C05468=1078.580,132.841,429.704,174.173,23.522,154.056
C05469=1078.585,133.090,429.683,174.174,23.524,154.056
C05470=1078.591,133.339,429.663,174.176,23.527,154.057
C05471=1078.596,133.588,429.643,174.178,23.529,154.057
C05472=1078.602,133.837,429.624,174.180,23.532,154.057
C05473=1078.607,134.086,429.603,174.181,23.533,154.057
C05474=1078.613,134.335,429.583,174.184,23.536,154.058
C05475=1078.619,134.584,429.563,174.186,23.538,154.058
C05476=1078.625,134.833,429.543,174.187,23.541,154.058
C05477=1078.630,135.083,429.522,174.190,23.543,154.058
C05478=1078.636,135.332,429.502,174.191,23.545,154.058
C05479=1078.642,135.581,429.482,174.193,23.548,154.058
C05480=1078.647,135.830,429.462,174.195,23.550,154.059
C05481=1078.653,136.079,429.442,174.197,23.552,154.059
C05482=1078.659,136.328,429.421,174.198,23.555,154.059
C05483=1078.664,136.578,429.402,174.201,23.557,154.059
C05484=1078.670,136.827,429.382,174.203,23.559,154.059
C05485=1078.676,137.075,429.362,174.204,23.561,154.060
C05486=1078.681,137.325,429.341,174.207,23.564,154.060
C05487=1078.687,137.574,429.321,174.208,23.566,154.060
C05488=1078.693,137.823,429.300,174.210,23.568,154.060
C05489=1078.699,138.072,429.280,174.212,23.571,154.061
C05490=1078.704,138.321,429.260,174.214,23.573,154.061
C05491=1078.710,138.570,429.240,174.215,23.575,154.061
C05492=1078.715,138.819,429.219,174.218,23.577,154.061
C05493=1078.720,139.068,429.199,174.220,23.580,154.061
C05494=1078.727,139.318,429.178,174.221,23.582,154.062
C05495=1078.732,139.567,429.158,174.224,23.584,154.062
C05496=1078.738,139.816,429.138,174.225,23.587,154.062
C05497=1078.744,140.065,429.117,174.228,23.589,154.062
C05498=1078.750,140.314,429.097,174.229,23.591,154.063
C05499=1078.755,140.563,429.077,174.231,23.594,154.063
C05500=1078.760,140.812,429.056,174.233,23.596,154.063
C05501=1078.767,141.061,429.036,174.235,23.598,154.063
C05502=1078.772,141.310,429.015,174.237,23.601,154.063
C05503=1078.777,141.560,428.995,174.239,23.603,154.064
C05504=1078.783,141.808,428.975,174.241,23.605,154.064
C05505=1078.788,142.058,428.954,174.243,23.608,154.064
C05506=1078.794,142.307,428.934,174.244,23.610,154.064
C05507=1078.800,142.557,428.913,174.247,23.612,154.064
C05508=1078.806,142.805,428.893,174.248,23.615,154.065
C05509=1078.812,143.086,428.869,174.251,23.617,154.065
C05510=1078.818,143.367,428.846,174.253,23.620,154.065
C05511=1078.824,143.647,428.824,174.255,23.622,154.065
C05512=1078.831,143.928,428.800,174.257,23.625,154.066
C05513=1078.836,144.177,428.779,174.260,23.627,154.066
C05514=1078.842,144.427,428.758,174.261,23.629,154.066
C05515=1078.848,144.675,428.738,174.263,23.632,154.066
C05516=1078.853,144.925,428.718,174.265,23.634,154.066
C05517=1078.859,145.173,428.697,174.267,23.637,154.067
C05518=1078.864,145.422,428.676,174.269,23.639,154.067
C05519=1078.871,145.672,428.656,174.271,23.641,154.067
C05520=1078.876,145.921,428.635,174.273,23.643,154.067
C05521=1078.881,146.169,428.614,174.274,23.645,154.067
C05522=1078.887,146.418,428.593,174.277,23.648,154.068
C05523=1078.893,146.668,428.573,174.279,23.650,154.068
C05524=1078.898,146.917,428.552,174.281,23.652,154.068
C05525=1078.904,147.166,428.531,174.283,23.655,154.068
C05526=1078.910,147.415,428.510,174.285,23.657,154.068
C05527=1078.916,147.664,428.490,174.286,23.659,154.069
C05528=1078.921,147.913,428.470,174.289,23.662,154.069
C05529=1078.927,148.162,428.448,174.290,23.663,154.069
C05530=1078.933,148.412,428.428,174.293,23.666,154.069
C05531=1078.938,148.661,428.407,174.295,23.668,154.069
C05532=1078.943,148.909,428.386,174.296,23.671,154.070
C05533=1078.949,149.158,428.365,174.299,23.673,154.070
C05534=1078.955,149.408,428.345,174.301,23.675,154.070
C05535=1078.961,149.656,428.324,174.302,23.677,154.070
C05536=1078.966,149.906,428.303,174.305,23.680,154.070
C05537=1078.972,150.155,428.281,174.306,23.682,154.071
C05538=1078.977,150.404,428.261,174.308,23.684,154.071
C05539=1078.983,150.653,428.240,174.311,23.687,154.071
C05540=1078.989,150.902,428.219,174.312,23.689,154.071
C05541=1078.994,151.151,428.198,174.314,23.691,154.071
C05542=1079.000,151.400,428.177,174.317,23.694,154.072
C05543=1079.005,151.649,428.156,174.318,23.696,154.072
C05544=1079.011,151.898,428.135,174.321,23.698,154.072
C05545=1079.016,152.147,428.114,174.323,23.701,154.072
C05546=1079.022,152.396,428.093,174.324,23.702,154.072
C05547=1079.028,152.646,428.072,174.326,23.705,154.073
C05548=1079.033,152.894,428.051,174.328,23.707,154.073
C05549=1079.039,153.143,428.030,174.330,23.709,154.073
C05550=1079.045,153.392,428.008,174.333,23.712,154.073
C05551=1079.050,153.642,427.988,174.334,23.714,154.073
C05552=1079.056,153.890,427.967,174.336,23.716,154.073
C05553=1079.061,154.140,427.946,174.339,23.719,154.074
C05554=1079.067,154.388,427.924,174.340,23.721,154.074
C05555=1079.073,154.638,427.904,174.342,23.723,154.074
C05556=1079.078,154.887,427.882,174.345,23.726,154.074
C05557=1079.084,155.135,427.861,174.346,23.727,154.074
C05558=1079.090,155.385,427.840,174.349,23.730,154.075
C05559=1079.095,155.634,427.819,174.351,23.732,154.075
C05560=1079.101,155.883,427.798,174.352,23.734,154.075
C05561=1079.107,156.132,427.777,174.354,23.737,154.075
C05562=1079.112,156.380,427.755,174.357,23.739,154.075
C05563=1079.117,156.631,427.734,174.358,23.741,154.076
C05564=1079.123,156.879,427.713,174.361,23.744,154.076
C05565=1079.129,157.128,427.691,174.363,23.746,154.076
C05566=1079.134,157.377,427.670,174.364,23.748,154.076
C05567=1079.140,157.626,427.649,174.367,23.751,154.076
C05568=1079.146,157.875,427.627,174.369,23.753,154.077
C05569=1079.151,158.124,427.607,174.371,23.755,154.077
C05570=1079.157,158.374,427.585,174.373,23.757,154.077
C05571=1079.162,158.622,427.563,174.375,23.760,154.077
C05572=1079.168,158.871,427.542,174.377,23.762,154.077
C05573=1079.175,159.152,427.518,174.380,23.764,154.078
C05574=1079.181,159.432,427.494,174.382,23.767,154.078
C05575=1079.187,159.712,427.471,174.384,23.769,154.078
C05576=1079.193,159.993,427.446,174.387,23.772,154.078
C05577=1079.199,160.242,427.425,174.388,23.774,154.078
C05578=1079.205,160.491,427.403,174.390,23.777,154.079
C05579=1079.211,160.740,427.382,174.393,23.779,154.079
C05580=1079.216,160.989,427.361,174.395,23.781,154.079
C05581=1079.222,161.238,427.339,174.396,23.784,154.079
C05582=1079.227,161.487,427.318,174.399,23.786,154.079
C05583=1079.233,161.736,427.296,174.401,23.788,154.080
C05584=1079.238,161.985,427.274,174.402,23.790,154.080
C05585=1079.244,162.234,427.253,174.405,23.793,154.080
C05586=1079.249,162.483,427.231,174.407,23.795,154.080
C05587=1079.255,162.732,427.209,174.409,23.797,154.080
C05588=1079.260,162.982,427.188,174.411,23.800,154.081
C05589=1079.265,163.230,427.167,174.413,23.802,154.081
C05590=1079.271,163.480,427.145,174.415,23.805,154.081
C05591=1079.276,163.728,427.123,174.417,23.807,154.081
C05592=1079.282,163.977,427.102,174.419,23.809,154.081
C05593=1079.287,164.226,427.080,174.422,23.812,154.082
C05594=1079.293,164.475,427.058,174.424,23.814,154.082
C05595=1079.298,164.724,427.036,174.425,23.816,154.082
C05596=1079.304,164.973,427.015,174.428,23.818,154.082
C05597=1079.309,165.222,426.993,174.430,23.821,154.082
C05598=1079.315,165.471,426.971,174.432,23.823,154.083
C05599=1079.320,165.721,426.949,174.434,23.825,154.083
C05600=1079.326,165.969,426.928,174.436,23.828,154.083
C05601=1079.331,166.219,426.906,174.438,23.830,154.083
C05602=1079.337,166.467,426.884,174.440,23.832,154.083
C05603=1079.342,166.717,426.862,174.442,23.835,154.084
C05604=1079.347,166.965,426.840,174.444,23.837,154.084
C05605=1079.353,167.215,426.819,174.447,23.840,154.084
C05606=1079.358,167.463,426.797,174.448,23.841,154.084
C05607=1079.364,167.712,426.774,174.450,23.844,154.084
C05608=1079.369,167.961,426.752,174.453,23.846,154.085
C05609=1079.375,168.210,426.731,174.455,23.848,154.085
C05610=1079.380,168.459,426.709,174.457,23.851,154.085
C05611=1079.386,168.708,426.687,174.459,23.853,154.085
C05612=1079.391,168.957,426.665,174.461,23.855,154.085
C05613=1079.397,169.206,426.644,174.464,23.858,154.086
C05614=1079.403,169.456,426.622,174.466,23.860,154.086
C05615=1079.408,169.704,426.599,174.467,23.863,154.086
C05616=1079.414,169.953,426.577,174.470,23.865,154.086
C05617=1079.419,170.202,426.556,174.472,23.867,154.086
C05618=1079.425,170.451,426.534,174.474,23.870,154.087
C05619=1079.431,170.700,426.512,174.476,23.871,154.087
C05620=1079.436,170.948,426.490,174.478,23.874,154.087
C05621=1079.442,171.198,426.467,174.480,23.876,154.087
C05622=1079.447,171.447,426.446,174.483,23.879,154.087
C05623=1079.453,171.696,426.424,174.484,23.880,154.087
C05624=1079.459,171.945,426.401,174.487,23.883,154.088
C05625=1079.464,172.193,426.380,174.489,23.885,154.088
C05626=1079.470,172.443,426.358,174.491,23.888,154.088
C05627=1079.475,172.691,426.335,174.494,23.890,154.088
C05628=1079.481,172.940,426.313,174.495,23.892,154.088
C05629=1079.486,173.190,426.291,174.497,23.894,154.089
C05630=1079.491,173.438,426.268,174.500,23.897,154.089
C05631=1079.498,173.687,426.247,174.502,23.899,154.089
C05632=1079.503,173.937,426.225,174.504,23.901,154.089
C05633=1079.509,174.185,426.203,174.506,23.903,154.089
C05634=1079.514,174.434,426.180,174.508,23.905,154.089
C05635=1079.520,174.684,426.158,174.511,23.908,154.090
C05636=1079.526,174.932,426.136,174.513,23.910,154.090
C05637=1079.532,175.212,426.111,174.515,23.913,154.090
C05638=1079.538,175.492,426.086,174.518,23.915,154.090
C05639=1079.545,175.773,426.061,174.520,23.918,154.091
C05640=1079.551,176.053,426.036,174.522,23.920,154.091
C05641=1079.557,176.302,426.013,174.525,23.922,154.091
C05642=1079.562,176.550,425.992,174.527,23.925,154.091
C05643=1079.568,176.800,425.969,174.529,23.927,154.091
C05644=1079.573,177.049,425.946,174.532,23.930,154.091
C05645=1079.579,177.298,425.925,174.533,23.931,154.092
C05646=1079.585,177.546,425.902,174.535,23.934,154.092
C05647=1079.590,177.795,425.880,174.538,23.936,154.092
C05648=1079.597,178.044,425.858,174.540,23.939,154.092
C05649=1079.602,178.293,425.835,174.543,23.941,154.092
C05650=1079.607,178.542,425.813,174.545,23.943,154.092
C05651=1079.614,178.790,425.791,174.546,23.945,154.093
C05652=1079.619,179.040,425.768,174.549,23.947,154.093
C05653=1079.625,179.289,425.745,174.551,23.950,154.093
C05654=1079.630,179.538,425.723,174.554,23.952,154.093
C05655=1079.636,179.786,425.701,174.556,23.955,154.093
C05656=1079.642,180.035,425.678,174.558,23.957,154.093
C05657=1079.647,180.285,425.656,174.560,23.959,154.094
C05658=1079.654,180.533,425.634,174.562,23.961,154.094
C05659=1079.659,180.783,425.611,174.564,23.963,154.094
C05660=1079.665,181.032,425.588,174.567,23.966,154.094
C05661=1079.670,181.280,425.566,174.569,23.968,154.094
C05662=1079.676,181.529,425.544,174.571,23.970,154.094
C05663=1079.682,181.778,425.521,174.574,23.972,154.095
C05664=1079.688,182.027,425.498,174.575,23.974,154.095
C05665=1079.693,182.276,425.476,174.578,23.976,154.095
C05666=1079.699,182.525,425.454,174.580,23.979,154.095
C05667=1079.705,182.774,425.431,174.582,23.981,154.095
C05668=1079.710,183.022,425.408,174.585,23.983,154.095
C05669=1079.716,183.271,425.386,174.587,23.986,154.096
C05670=1079.721,183.520,425.363,174.590,23.988,154.096
C05671=1079.728,183.769,425.341,174.592,23.990,154.096
C05672=1079.734,184.018,425.318,174.594,23.992,154.096
C05673=1079.739,184.267,425.296,174.596,23.995,154.096
C05674=1079.745,184.516,425.273,174.598,23.997,154.096
C05675=1079.751,184.765,425.250,174.601,23.999,154.097
C05676=1079.757,185.014,425.227,174.603,24.001,154.097
C05677=1079.763,185.263,425.204,174.605,24.003,154.097
C05678=1079.767,185.511,425.181,174.608,24.006,154.097
C05679=1079.773,185.761,425.159,174.610,24.008,154.097
C05680=1079.778,186.010,425.136,174.611,24.011,154.098
C05681=1079.784,186.258,425.113,174.614,24.013,154.098
C05682=1079.790,186.507,425.090,174.616,24.015,154.098
C05683=1079.795,186.756,425.068,174.618,24.018,154.098
C05684=1079.800,187.005,425.044,174.621,24.020,154.098
C05685=1079.806,187.254,425.021,174.623,24.023,154.099
C05686=1079.811,187.503,424.998,174.625,24.025,154.099
C05687=1079.817,187.751,424.975,174.628,24.027,154.099
C05688=1079.823,188.000,424.952,174.630,24.030,154.099
C05689=1079.827,188.249,424.929,174.633,24.032,154.099
C05690=1079.833,188.498,424.906,174.634,24.034,154.099
C05691=1079.839,188.747,424.883,174.636,24.036,154.100
C05692=1079.844,188.996,424.860,174.639,24.039,154.100
C05693=1079.850,189.244,424.837,174.641,24.041,154.100
C05694=1079.855,189.494,424.814,174.643,24.044,154.100
C05695=1079.861,189.743,424.791,174.646,24.046,154.100
C05696=1079.867,189.991,424.768,174.648,24.048,154.101
C05697=1079.872,190.240,424.745,174.650,24.051,154.101
C05698=1079.877,190.488,424.722,174.653,24.053,154.101
C05699=1079.882,190.738,424.699,174.655,24.055,154.101
C05700=1079.888,190.987,424.676,174.657,24.058,154.101
C05701=1079.895,191.267,424.650,174.660,24.060,154.102
C05702=1079.901,191.546,424.624,174.662,24.063,154.102
C05703=1079.907,191.827,424.597,174.665,24.066,154.102
C05704=1079.913,192.106,424.571,174.668,24.068,154.102
C05705=1079.919,192.355,424.548,174.670,24.070,154.102
C05706=1079.925,192.604,424.526,174.672,24.073,154.103
C05707=1079.930,192.853,424.502,174.675,24.075,154.103
C05708=1079.936,193.101,424.478,174.677,24.077,154.103
C05709=1079.941,193.350,424.455,174.679,24.080,154.103
C05710=1079.947,193.599,424.432,174.681,24.082,154.103
C05711=1079.952,193.848,424.409,174.683,24.084,154.103
C05712=1079.958,194.097,424.386,174.686,24.087,154.104
C05713=1079.964,194.345,424.362,174.688,24.089,154.104
C05714=1079.969,194.595,424.339,174.690,24.091,154.104
C05715=1079.975,194.844,424.316,174.693,24.093,154.104
C05716=1079.980,195.092,424.293,174.695,24.096,154.104
C05717=1079.986,195.341,424.269,174.697,24.098,154.105
C05718=1079.991,195.590,424.246,174.700,24.100,154.105
C05719=1079.997,195.839,424.223,174.702,24.103,154.105
C05720=1080.003,196.087,424.199,174.704,24.105,154.105
C05721=1080.008,196.336,424.175,174.707,24.107,154.105
C05722=1080.014,196.585,424.153,174.709,24.110,154.105
C05723=1080.020,196.833,424.129,174.712,24.112,154.106
C05724=1080.025,197.083,424.105,174.714,24.114,154.106
C05725=1080.031,197.332,424.082,174.716,24.117,154.106
C05726=1080.037,197.581,424.058,174.719,24.119,154.106
C05727=1080.042,197.830,424.035,174.721,24.121,154.106
C05728=1080.048,198.079,424.012,174.723,24.124,154.107
C05729=1080.054,198.327,423.988,174.726,24.126,154.107
C05730=1080.059,198.576,423.965,174.728,24.128,154.107
C05731=1080.065,198.824,423.941,174.731,24.131,154.107
C05732=1080.071,199.073,423.918,174.733,24.133,154.107
C05733=1080.076,199.322,423.894,174.735,24.135,154.107
C05734=1080.082,199.571,423.871,174.738,24.137,154.108
C05735=1080.087,199.821,423.847,174.740,24.140,154.108
C05736=1080.093,200.069,423.823,174.742,24.142,154.108
C05737=1080.099,200.318,423.800,174.745,24.144,154.108
C05738=1080.104,200.566,423.776,174.747,24.147,154.108
C05739=1080.110,200.815,423.753,174.749,24.149,154.108
C05740=1080.116,201.064,423.729,174.752,24.151,154.109
C05741=1080.122,201.313,423.705,174.754,24.154,154.109
C05742=1080.128,201.562,423.682,174.757,24.156,154.109
C05743=1080.133,201.810,423.658,174.759,24.159,154.109
C05744=1080.139,202.059,423.635,174.761,24.161,154.109
C05745=1080.144,202.308,423.610,174.764,24.163,154.109
C05746=1080.151,202.557,423.587,174.766,24.165,154.110
C05747=1080.156,202.806,423.563,174.768,24.168,154.110
C05748=1080.162,203.054,423.539,174.771,24.170,154.110
C05749=1080.167,203.304,423.516,174.773,24.172,154.110
C05750=1080.173,203.552,423.492,174.776,24.175,154.110
C05751=1080.178,203.800,423.468,174.778,24.177,154.111
C05752=1080.184,204.050,423.444,174.780,24.179,154.111
C05753=1080.190,204.299,423.420,174.783,24.182,154.111
C05754=1080.195,204.547,423.396,174.785,24.184,154.111
C05755=1080.200,204.796,423.372,174.787,24.186,154.111
C05756=1080.206,205.045,423.349,174.791,24.189,154.112
C05757=1080.211,205.293,423.324,174.793,24.192,154.112
C05758=1080.217,205.543,423.300,174.795,24.194,154.112
C05759=1080.223,205.791,423.277,174.798,24.196,154.112
C05760=1080.228,206.040,423.253,174.800,24.199,154.112
C05761=1080.234,206.289,423.228,174.803,24.201,154.112
C05762=1080.240,206.538,423.204,174.805,24.203,154.113
C05763=1080.245,206.787,423.181,174.807,24.206,154.113
C05764=1080.251,207.035,423.157,174.809,24.208,154.113
C05765=1080.274,208.069,423.057,174.909,24.261,154.111
C05766=1080.283,208.468,423.017,174.913,24.267,154.112
C05767=1080.292,208.867,422.978,174.917,24.272,154.113
C05768=1080.302,209.266,422.939,174.921,24.277,154.113
C05769=1080.311,209.665,422.899,174.924,24.282,154.114
C05770=1080.317,209.914,422.874,174.926,24.286,154.114
C05771=1080.322,210.163,422.850,174.929,24.289,154.115
C05772=1080.328,210.411,422.825,174.931,24.293,154.115
C05773=1080.334,210.660,422.800,174.934,24.296,154.116
C05774=1080.339,210.909,422.776,174.936,24.299,154.116
C05775=1080.345,211.157,422.751,174.938,24.303,154.116
C05776=1080.351,211.406,422.726,174.940,24.306,154.117
C05777=1080.356,211.655,422.702,174.943,24.309,154.117
C05778=1080.362,211.904,422.677,174.945,24.313,154.118
C05779=1080.368,212.152,422.652,174.947,24.316,154.118
C05780=1080.373,212.401,422.626,174.949,24.319,154.118
C05781=1080.378,212.650,422.602,174.952,24.323,154.119
C05782=1080.385,212.899,422.577,174.954,24.326,154.119
C05783=1080.391,213.148,422.552,174.957,24.329,154.120
C05784=1080.396,213.396,422.528,174.959,24.332,154.120
C05785=1080.402,213.645,422.503,174.961,24.336,154.121
C05786=1080.407,213.894,422.478,174.964,24.340,154.121
C05787=1080.413,214.143,422.452,174.966,24.343,154.121
C05788=1080.418,214.391,422.427,174.968,24.346,154.122
C05789=1080.424,214.640,422.403,174.970,24.349,154.122
C05790=1080.430,214.888,422.378,174.973,24.353,154.122
C05791=1080.436,215.137,422.353,174.975,24.356,154.123
C05792=1080.441,215.385,422.328,174.977,24.359,154.123
C05793=1080.447,215.635,422.303,174.979,24.362,154.124
C05794=1080.453,215.883,422.278,174.982,24.366,154.124
C05795=1080.458,216.131,422.253,174.984,24.370,154.125
C05796=1080.464,216.381,422.228,174.986,24.373,154.125
C05797=1080.469,216.629,422.203,174.989,24.376,154.125
C05798=1080.475,216.878,422.178,174.992,24.380,154.126
C05799=1080.481,217.127,422.153,174.994,24.383,154.126
C05800=1080.486,217.375,422.127,174.996,24.386,154.127
C05801=1080.492,217.624,422.102,174.998,24.389,154.127
C05802=1080.498,217.872,422.077,175.001,24.393,154.127
C05803=1080.504,218.121,422.052,175.003,24.396,154.128
C05804=1080.509,218.370,422.026,175.005,24.399,154.128
C05805=1080.515,218.619,422.002,175.007,24.402,154.129
C05806=1080.521,218.867,421.977,175.010,24.406,154.129
C05807=1080.526,219.116,421.951,175.013,24.409,154.129
C05808=1080.532,219.364,421.926,175.015,24.412,154.130
C05809=1080.538,219.614,421.901,175.018,24.416,154.130
C05810=1080.544,219.862,421.876,175.020,24.420,154.131
C05811=1080.549,220.111,421.850,175.022,24.423,154.131
C05812=1080.555,220.359,421.825,175.024,24.426,154.132
C05813=1080.561,220.608,421.799,175.027,24.430,154.132
C05814=1080.567,220.857,421.774,175.029,24.433,154.132
C05815=1080.572,221.105,421.749,175.031,24.436,154.133
C05816=1080.578,221.354,421.724,175.033,24.439,154.133
C05817=1080.584,221.603,421.698,175.036,24.443,154.133
C05818=1080.593,222.006,421.657,175.040,24.448,154.134
C05819=1080.602,222.409,421.615,175.044,24.453,154.135
C05820=1080.612,222.813,421.574,175.048,24.459,154.135
C05821=1080.621,223.215,421.533,175.052,24.464,154.136
C05822=1080.626,223.464,421.507,175.054,24.467,154.136
C05823=1080.632,223.713,421.482,175.057,24.471,154.137
C05824=1080.637,223.961,421.456,175.059,24.474,154.137
C05825=1080.643,224.210,421.431,175.061,24.478,154.138
C05826=1080.649,224.459,421.405,175.064,24.481,154.138
C05827=1080.655,224.707,421.379,175.066,24.484,154.139
C05828=1080.660,224.956,421.354,175.068,24.488,154.139
C05829=1080.666,225.204,421.328,175.071,24.491,154.139
C05830=1080.672,225.453,421.303,175.073,24.494,154.140
C05831=1080.677,225.702,421.277,175.075,24.498,154.140
C05832=1080.683,225.950,421.252,175.078,24.501,154.141
C05833=1080.688,226.199,421.226,175.081,24.504,154.141
C05834=1080.694,226.448,421.200,175.083,24.508,154.142
C05835=1080.700,226.697,421.174,175.085,24.511,154.142
C05836=1080.706,226.945,421.148,175.088,24.515,154.142
C05837=1080.711,227.193,421.123,175.090,24.518,154.143
C05838=1080.717,227.442,421.097,175.092,24.521,154.143
C05839=1080.723,227.691,421.072,175.095,24.525,154.143
C05840=1080.728,227.940,421.046,175.097,24.528,154.144
C05841=1080.735,228.188,421.020,175.099,24.531,154.144
C05842=1080.740,228.437,420.994,175.102,24.535,154.145
C05843=1080.746,228.686,420.968,175.105,24.538,154.145
C05844=1080.751,228.934,420.943,175.107,24.541,154.145
C05845=1080.757,229.182,420.916,175.110,24.545,154.146
C05846=1080.763,229.431,420.890,175.112,24.548,154.146
C05847=1080.769,229.680,420.865,175.114,24.551,154.147
C05848=1080.774,229.929,420.839,175.117,24.554,154.147
C05849=1080.780,230.177,420.812,175.119,24.558,154.147
C05850=1080.786,230.426,420.787,175.121,24.561,154.148
C05851=1080.792,230.675,420.761,175.124,24.564,154.148
C05852=1080.797,230.922,420.735,175.127,24.568,154.149
C05853=1080.802,231.171,420.709,175.129,24.571,154.149
C05854=1080.809,231.420,420.683,175.132,24.575,154.150
C05855=1080.814,231.668,420.657,175.134,24.578,154.150
C05856=1080.820,231.917,420.631,175.136,24.581,154.150
C05857=1080.826,232.166,420.604,175.139,24.585,154.151
C05858=1080.831,232.415,420.578,175.141,24.588,154.151
C05859=1080.837,232.663,420.552,175.143,24.591,154.152
C05860=1080.843,232.912,420.526,175.146,24.595,154.152
C05861=1080.849,233.160,420.500,175.148,24.598,154.152
C05862=1080.854,233.409,420.474,175.151,24.601,154.153
C05863=1080.859,233.657,420.448,175.154,24.605,154.153
C05864=1080.865,233.906,420.421,175.156,24.608,154.154
C05865=1080.871,234.154,420.395,175.159,24.612,154.154
C05866=1080.876,234.403,420.369,175.161,24.615,154.154
C05867=1080.882,234.651,420.342,175.163,24.618,154.155
C05868=1080.888,234.900,420.317,175.166,24.622,154.155
C05869=1080.894,235.148,420.290,175.168,24.625,154.156
C05870=1080.903,235.543,420.248,175.172,24.630,154.156
C05871=1080.911,235.938,420.207,175.176,24.636,154.157
C05872=1080.921,236.333,420.165,175.180,24.641,154.158
C05873=1080.930,236.728,420.122,175.184,24.646,154.158
C05874=1080.935,236.976,420.096,175.187,24.650,154.159
C05875=1080.941,237.225,420.070,175.189,24.653,154.159
C05876=1080.947,237.474,420.043,175.192,24.657,154.160
C05877=1080.952,237.722,420.017,175.194,24.660,154.160
C05878=1080.958,237.971,419.991,175.196,24.663,154.160
C05879=1080.964,238.219,419.964,175.199,24.667,154.161
C05880=1080.969,238.468,419.937,175.201,24.670,154.161
C05881=1080.975,238.716,419.911,175.204,24.673,154.162
C05882=1080.981,238.965,419.885,175.206,24.677,154.162
C05883=1080.986,239.213,419.858,175.209,24.680,154.162
C05884=1080.992,239.462,419.831,175.212,24.683,154.163
C05885=1080.998,239.710,419.805,175.214,24.686,154.163
C05886=1081.004,239.958,419.778,175.217,24.690,154.164
C05887=1081.009,240.207,419.752,175.219,24.694,154.164
C05888=1081.016,240.456,419.725,175.221,24.697,154.165
C05889=1081.021,240.705,419.699,175.224,24.700,154.165
C05890=1081.027,240.953,419.672,175.226,24.704,154.165
C05891=1081.033,241.201,419.645,175.229,24.707,154.166
C05892=1081.038,241.450,419.618,175.231,24.710,154.166
C05893=1081.044,241.698,419.591,175.234,24.714,154.166
C05894=1081.050,241.947,419.565,175.237,24.717,154.167
C05895=1081.055,242.195,419.538,175.239,24.720,154.167
C05896=1081.061,242.444,419.511,175.242,24.724,154.168
C05897=1081.067,242.693,419.484,175.244,24.727,154.168
C05898=1081.073,242.941,419.458,175.247,24.730,154.168
C05899=1081.078,243.190,419.431,175.249,24.734,154.169
C05900=1081.084,243.438,419.404,175.252,24.738,154.169
C05901=1081.090,243.686,419.377,175.254,24.741,154.170
C05902=1081.096,243.935,419.351,175.256,24.744,154.170
C05903=1081.101,244.183,419.323,175.260,24.747,154.171
C05904=1081.106,244.432,419.297,175.262,24.751,154.171
C05905=1081.113,244.681,419.270,175.265,24.755,154.172
C05906=1081.118,244.930,419.242,175.267,24.758,154.172
C05907=1081.124,245.178,419.216,175.270,24.761,154.172
C05908=1081.129,245.426,419.189,175.272,24.764,154.173
C05909=1081.134,245.675,419.162,175.274,24.768,154.173
C05910=1081.140,245.923,419.135,175.277,24.771,154.174
C05911=1081.147,246.172,419.108,175.279,24.775,154.174
C05912=1081.152,246.420,419.080,175.282,24.778,154.174
C05913=1081.158,246.669,419.054,175.284,24.781,154.175
C05914=1081.163,246.917,419.027,175.288,24.785,154.175
C05915=1081.168,247.166,419.000,175.290,24.788,154.176
C05916=1081.175,247.413,418.972,175.293,24.792,154.176
C05917=1081.180,247.663,418.945,175.295,24.795,154.177
C05918=1081.186,247.911,418.918,175.297,24.799,154.177
C05919=1081.191,248.160,418.891,175.300,24.802,154.177
C05920=1081.197,248.408,418.864,175.302,24.805,154.178
C05921=1081.202,248.656,418.836,175.305,24.809,154.178
C05922=1081.211,249.044,418.794,175.309,24.814,154.179
C05923=1081.220,249.432,418.752,175.313,24.820,154.180
C05924=1081.228,249.820,418.709,175.317,24.825,154.180
C05925=1081.238,250.208,418.666,175.321,24.830,154.181
C05926=1081.243,250.457,418.639,175.324,24.834,154.181
C05927=1081.249,250.705,418.611,175.326,24.837,154.182
C05928=1081.254,250.954,418.584,175.329,24.841,154.182
C05929=1081.260,251.201,418.557,175.331,24.844,154.183
C05930=1081.266,251.451,418.529,175.334,24.848,154.183
C05931=1081.271,251.700,418.502,175.336,24.851,154.184
C05932=1081.277,251.947,418.474,175.339,24.855,154.184
C05933=1081.282,252.196,418.447,175.341,24.858,154.184
C05934=1081.289,252.444,418.419,175.344,24.862,154.185
C05935=1081.294,252.693,418.392,175.347,24.865,154.185
C05936=1081.299,252.941,418.364,175.350,24.869,154.186
C05937=1081.306,253.190,418.337,175.352,24.872,154.186
C05938=1081.311,253.438,418.309,175.355,24.875,154.186
C05939=1081.317,253.686,418.282,175.357,24.878,154.187
C05940=1081.323,253.935,418.254,175.360,24.883,154.187
C05941=1081.328,254.183,418.226,175.362,24.886,154.188
C05942=1081.334,254.432,418.200,175.365,24.889,154.188
C05943=1081.340,254.681,418.171,175.367,24.892,154.189
C05944=1081.345,254.929,418.143,175.370,24.896,154.189
C05945=1081.351,255.177,418.117,175.373,24.899,154.189
C05946=1081.357,255.426,418.088,175.376,24.903,154.190
C05947=1081.363,255.673,418.061,175.378,24.906,154.190
C05948=1081.368,255.922,418.034,175.381,24.910,154.191
C05949=1081.374,256.171,418.005,175.383,24.913,154.191
C05950=1081.380,256.419,417.978,175.386,24.916,154.191
C05951=1081.386,256.668,417.950,175.388,24.920,154.192
C05952=1081.391,256.916,417.922,175.391,24.923,154.192
C05953=1081.397,257.164,417.895,175.393,24.927,154.193
C05954=1081.403,257.412,417.867,175.396,24.930,154.193
C05955=1081.408,257.661,417.840,175.399,24.933,154.194
C05956=1081.414,257.910,417.811,175.402,24.937,154.194
C05957=1081.420,258.158,417.784,175.404,24.940,154.195
C05958=1081.426,258.406,417.756,175.407,24.944,154.195
C05959=1081.431,258.654,417.728,175.409,24.947,154.195
C05960=1081.438,258.903,417.700,175.412,24.951,154.196
C05961=1081.443,259.152,417.673,175.415,24.954,154.196
C05962=1081.449,259.400,417.644,175.417,24.957,154.197
C05963=1081.454,259.648,417.616,175.420,24.961,154.197
C05964=1081.461,259.897,417.589,175.423,24.964,154.197
C05965=1081.466,260.145,417.561,175.426,24.968,154.198
C05966=1081.472,260.394,417.532,175.428,24.971,154.198
C05967=1081.478,260.642,417.504,175.431,24.975,154.199
C05968=1081.484,260.890,417.477,175.433,24.978,154.199
C05969=1081.490,261.138,417.449,175.436,24.982,154.200
C05970=1081.496,261.387,417.420,175.438,24.985,154.200
C05971=1081.501,261.635,417.392,175.441,24.988,154.200
C05972=1081.508,261.883,417.365,175.444,24.992,154.201
C05973=1081.513,262.131,417.337,175.447,24.995,154.201
C05974=1081.522,262.517,417.293,175.451,25.001,154.202
C05975=1081.531,262.903,417.249,175.455,25.006,154.202
C05976=1081.540,263.287,417.205,175.459,25.011,154.203
C05977=1081.550,263.673,417.162,175.463,25.016,154.204
C05978=1081.556,263.921,417.134,175.466,25.020,154.204
C05979=1081.561,264.169,417.106,175.468,25.023,154.205
C05980=1081.567,264.418,417.078,175.471,25.026,154.205
C05981=1081.573,264.666,417.049,175.474,25.030,154.206
C05982=1081.579,264.914,417.021,175.477,25.034,154.206
C05983=1081.584,265.162,416.993,175.480,25.037,154.206
C05984=1081.590,265.411,416.964,175.482,25.041,154.207
C05985=1081.596,265.659,416.936,175.485,25.044,154.207
C05986=1081.602,265.907,416.907,175.487,25.047,154.208
C05987=1081.607,266.156,416.879,175.490,25.051,154.208
C05988=1081.612,266.404,416.851,175.492,25.054,154.209
C05989=1081.618,266.653,416.822,175.495,25.058,154.209
C05990=1081.624,266.901,416.794,175.498,25.062,154.209
C05991=1081.630,267.149,416.765,175.500,25.065,154.210
C05992=1081.636,267.398,416.736,175.504,25.069,154.210
C05993=1081.641,267.646,416.708,175.506,25.072,154.211
C05994=1081.647,267.894,416.680,175.509,25.076,154.211
C05995=1081.653,268.142,416.651,175.512,25.079,154.212
C05996=1081.659,268.390,416.623,175.514,25.083,154.212
C05997=1081.665,268.639,416.595,175.517,25.086,154.213
C05998=1081.670,268.887,416.565,175.519,25.089,154.213
C05999=1081.676,269.136,416.537,175.522,25.093,154.213
C06000=1081.682,269.384,416.508,175.525,25.097,154.214
C06001=1081.687,269.632,416.480,175.527,25.100,154.214
C06002=1081.693,269.880,416.451,175.531,25.103,154.215
C06003=1081.699,270.129,416.423,175.533,25.107,154.215
C06004=1081.704,270.377,416.393,175.536,25.111,154.216
C06005=1081.710,270.625,416.365,175.539,25.115,154.216
C06006=1081.716,270.873,416.336,175.541,25.118,154.217
C06007=1081.722,271.121,416.308,175.544,25.121,154.217
C06008=1081.727,271.370,416.278,175.546,25.125,154.217
C06009=1081.733,271.619,416.250,175.549,25.128,154.218
C06010=1081.739,271.867,416.221,175.552,25.132,154.218
C06011=1081.745,272.115,416.193,175.554,25.135,154.219
C06012=1081.750,272.363,416.163,175.558,25.139,154.219
C06013=1081.757,272.611,416.134,175.561,25.142,154.220
C06014=1081.762,272.859,416.106,175.563,25.146,154.220
C06015=1081.767,273.108,416.077,175.566,25.149,154.220
C06016=1081.774,273.356,416.048,175.568,25.153,154.221
C06017=1081.780,273.605,416.019,175.571,25.157,154.221
C06018=1081.785,273.853,415.990,175.574,25.160,154.222
C06019=1081.791,274.101,415.961,175.576,25.164,154.222
C06020=1081.797,274.349,415.932,175.579,25.167,154.223
C06021=1081.802,274.598,415.903,175.582,25.171,154.223
C06022=1081.808,274.845,415.875,175.584,25.174,154.224
C06023=1081.813,275.094,415.845,175.587,25.178,154.224
C06024=1081.820,275.342,415.816,175.591,25.182,154.225
C06025=1081.826,275.591,415.788,175.593,25.185,154.225
C06026=1081.834,275.978,415.742,175.597,25.191,154.226
C06027=1081.843,276.366,415.696,175.602,25.196,154.226
C06028=1081.853,276.755,415.650,175.605,25.202,154.227
C06029=1081.860,277.143,415.605,175.610,25.207,154.228
C06030=1081.867,277.391,415.576,175.613,25.211,154.228
C06031=1081.872,277.640,415.546,175.615,25.214,154.229
C06032=1081.879,277.888,415.517,175.618,25.218,154.229
C06033=1081.883,278.136,415.488,175.621,25.222,154.230
C06034=1081.890,278.384,415.459,175.623,25.226,154.230
C06035=1081.895,278.632,415.429,175.627,25.229,154.231
C06036=1081.901,278.881,415.400,175.630,25.233,154.231
C06037=1081.907,279.129,415.371,175.632,25.236,154.232
C06038=1081.913,279.377,415.342,175.635,25.240,154.232
C06039=1081.919,279.626,415.312,175.638,25.244,154.233
C06040=1081.924,279.873,415.283,175.640,25.247,154.233
C06041=1081.930,280.121,415.254,175.643,25.251,154.233
C06042=1081.935,280.370,415.224,175.646,25.255,154.234
C06043=1081.942,280.618,415.195,175.648,25.258,154.234
C06044=1081.947,280.866,415.165,175.651,25.261,154.235
C06045=1081.954,281.114,415.136,175.654,25.265,154.235
C06046=1081.959,281.362,415.106,175.656,25.269,154.236
C06047=1081.965,281.611,415.076,175.660,25.272,154.236
C06048=1081.971,281.859,415.047,175.663,25.276,154.237
C06049=1081.976,282.107,415.018,175.665,25.279,154.237
C06050=1081.982,282.354,414.988,175.668,25.283,154.238
C06051=1081.987,282.603,414.958,175.671,25.287,154.238
C06052=1081.993,282.851,414.929,175.674,25.291,154.239
C06053=1081.999,283.100,414.899,175.676,25.294,154.239
C06054=1082.004,283.348,414.870,175.679,25.298,154.240
C06055=1082.010,283.596,414.839,175.682,25.302,154.240
C06056=1082.017,283.844,414.810,175.684,25.305,154.241
C06057=1082.022,284.092,414.781,175.687,25.309,154.241
C06058=1082.028,284.340,414.750,175.690,25.313,154.242
C06059=1082.033,284.589,414.721,175.693,25.316,154.242
C06060=1082.039,284.837,414.691,175.696,25.320,154.242
C06061=1082.045,285.085,414.661,175.699,25.324,154.243
C06062=1082.051,285.333,414.632,175.702,25.327,154.243
C06063=1082.056,285.581,414.602,175.704,25.331,154.244
C06064=1082.062,285.829,414.572,175.707,25.335,154.244
C06065=1082.068,286.078,414.542,175.710,25.338,154.245
C06066=1082.074,286.325,414.512,175.713,25.342,154.245
C06067=1082.080,286.574,414.483,175.715,25.345,154.246
C06068=1082.086,286.821,414.452,175.718,25.349,154.246
C06069=1082.091,287.070,414.423,175.721,25.353,154.247
C06070=1082.097,287.318,414.392,175.723,25.356,154.247
C06071=1082.103,287.566,414.363,175.726,25.360,154.248
C06072=1082.109,287.814,414.333,175.729,25.364,154.248
C06073=1082.115,288.062,414.303,175.732,25.368,154.249
C06074=1082.120,288.310,414.273,175.735,25.371,154.249
C06075=1082.126,288.558,414.243,175.738,25.375,154.250
C06076=1082.132,288.806,414.213,175.741,25.379,154.250
C06077=1082.137,289.055,414.183,175.744,25.383,154.251
C06078=1082.147,289.453,414.135,175.748,25.388,154.251
C06079=1082.156,289.850,414.086,175.753,25.395,154.252
C06080=1082.166,290.248,414.038,175.757,25.400,154.253
C06081=1082.174,290.646,413.990,175.762,25.406,154.254
C06082=1082.180,290.894,413.960,175.764,25.410,154.254
C06083=1082.186,291.142,413.929,175.767,25.413,154.255
C06084=1082.192,291.390,413.900,175.770,25.417,154.255
C06085=1082.198,291.639,413.869,175.773,25.421,154.256
C06086=1082.204,291.887,413.839,175.776,25.425,154.256
C06087=1082.210,292.135,413.808,175.778,25.428,154.257
C06088=1082.215,292.382,413.778,175.781,25.432,154.257
C06089=1082.221,292.631,413.748,175.784,25.436,154.258
C06090=1082.227,292.879,413.718,175.787,25.440,154.258
C06091=1082.233,293.126,413.688,175.790,25.443,154.259
C06092=1082.238,293.374,413.657,175.793,25.447,154.259
C06093=1082.244,293.623,413.626,175.796,25.451,154.260
C06094=1082.250,293.871,413.596,175.799,25.455,154.260
C06095=1082.256,294.119,413.565,175.802,25.459,154.261
C06096=1082.261,294.367,413.536,175.804,25.463,154.261
C06097=1082.267,294.615,413.505,175.807,25.466,154.262
C06098=1082.273,294.863,413.475,175.810,25.470,154.262
C06099=1082.279,295.111,413.444,175.813,25.474,154.263
C06100=1082.285,295.359,413.414,175.816,25.478,154.263
C06101=1082.290,295.607,413.383,175.818,25.482,154.264
C06102=1082.296,295.855,413.353,175.821,25.485,154.264
C06103=1082.302,296.103,413.322,175.824,25.489,154.265
C06104=1082.308,296.351,413.292,175.827,25.493,154.265
C06105=1082.313,296.600,413.261,175.830,25.497,154.266
C06106=1082.319,296.847,413.230,175.832,25.500,154.266
C06107=1082.325,297.095,413.199,175.835,25.504,154.267
C06108=1082.332,297.343,413.168,175.838,25.508,154.267
C06109=1082.337,297.591,413.138,175.841,25.512,154.268
C06110=1082.343,297.839,413.107,175.844,25.516,154.268
C06111=1082.348,298.087,413.077,175.847,25.520,154.269
C06112=1082.354,298.336,413.045,175.850,25.524,154.270
C06113=1082.360,298.584,413.015,175.853,25.528,154.270
C06114=1082.365,298.831,412.983,175.856,25.532,154.271
C06115=1082.371,299.079,412.953,175.859,25.536,154.271
C06116=1082.376,299.327,412.922,175.862,25.539,154.272
C06117=1082.383,299.576,412.891,175.864,25.543,154.272
C06118=1082.388,299.823,412.860,175.867,25.547,154.273
C06119=1082.394,300.071,412.829,175.870,25.551,154.273
C06120=1082.399,300.319,412.799,175.873,25.555,154.274
C06121=1082.405,300.567,412.768,175.876,25.559,154.274
C06122=1082.411,300.815,412.736,175.879,25.563,154.275
C06123=1082.417,301.063,412.706,175.881,25.567,154.276
C06124=1082.422,301.311,412.675,175.884,25.571,154.276
C06125=1082.428,301.559,412.643,175.887,25.575,154.277
C06126=1082.433,301.807,412.612,175.890,25.579,154.277
C06127=1082.440,302.054,412.581,175.893,25.582,154.278
C06128=1082.445,302.302,412.550,175.896,25.586,154.278
C06129=1082.451,302.551,412.520,175.899,25.590,154.279
C06130=1082.461,302.963,412.467,175.904,25.597,154.280
C06131=1082.470,303.375,412.416,175.908,25.603,154.280
C06132=1082.479,303.787,412.364,175.913,25.610,154.281
C06133=1082.489,304.199,412.312,175.918,25.616,154.282
C06134=1082.494,304.447,412.281,175.921,25.621,154.283
C06135=1082.501,304.695,412.250,175.924,25.625,154.283
C06136=1082.506,304.943,412.218,175.927,25.629,154.284
C06137=1082.512,305.191,412.188,175.930,25.632,154.285
C06138=1082.518,305.439,412.156,175.933,25.636,154.285
C06139=1082.523,305.687,412.125,175.936,25.640,154.286
C06140=1082.530,305.935,412.093,175.939,25.644,154.286
C06141=1082.535,306.182,412.062,175.941,25.648,154.287
C06142=1082.541,306.431,412.031,175.944,25.652,154.287
C06143=1082.547,306.678,411.999,175.947,25.656,154.288
C06144=1082.552,306.926,411.968,175.950,25.660,154.288
C06145=1082.559,307.174,411.937,175.953,25.664,154.289
C06146=1082.564,307.422,411.905,175.956,25.668,154.290
C06147=1082.570,307.670,411.873,175.959,25.672,154.290
C06148=1082.576,307.917,411.842,175.962,25.676,154.291
C06149=1082.582,308.166,411.811,175.965,25.680,154.291
C06150=1082.587,308.414,411.779,175.968,25.684,154.292
C06151=1082.594,308.662,411.748,175.970,25.688,154.292
C06152=1082.599,308.909,411.716,175.973,25.692,154.293
C06153=1082.605,309.157,411.684,175.976,25.696,154.293
C06154=1082.611,309.405,411.654,175.979,25.700,154.294
C06155=1082.617,309.653,411.622,175.982,25.704,154.294
C06156=1082.623,309.902,411.590,175.985,25.708,154.295
C06157=1082.629,310.149,411.558,175.988,25.712,154.296
C06158=1082.635,310.397,411.526,175.991,25.716,154.296
C06159=1082.641,310.644,411.495,175.994,25.720,154.297
C06160=1082.647,310.893,411.463,175.997,25.724,154.297
C06161=1082.653,311.140,411.432,176.000,25.728,154.298
C06162=1082.659,311.388,411.400,176.003,25.732,154.298
C06163=1082.665,311.636,411.368,176.007,25.736,154.299
C06164=1082.670,311.884,411.336,176.009,25.740,154.300
C06165=1082.677,312.132,411.305,176.012,25.744,154.300
C06166=1082.683,312.380,411.273,176.015,25.748,154.301
C06167=1082.688,312.627,411.241,176.018,25.752,154.301
C06168=1082.694,312.876,411.209,176.021,25.756,154.302
C06169=1082.700,313.124,411.177,176.024,25.760,154.302
C06170=1082.706,313.371,411.146,176.027,25.764,154.303
C06171=1082.712,313.619,411.114,176.030,25.768,154.304
C06172=1082.718,313.867,411.082,176.033,25.772,154.304
C06173=1082.724,314.115,411.050,176.036,25.776,154.305
C06174=1082.730,314.363,411.018,176.039,25.781,154.305
C06175=1082.737,314.610,410.986,176.042,25.785,154.306
C06176=1082.743,314.859,410.954,176.045,25.788,154.306
C06177=1082.748,315.106,410.922,176.048,25.793,154.307
C06178=1082.753,315.355,410.890,176.051,25.797,154.308
C06179=1082.759,315.602,410.858,176.054,25.801,154.308
C06180=1082.765,315.850,410.825,176.057,25.805,154.309
C06181=1082.771,316.098,410.793,176.060,25.810,154.309
C06182=1082.781,316.513,410.739,176.064,25.816,154.310
C06183=1082.790,316.928,410.685,176.069,25.824,154.312
C06184=1082.799,317.344,410.631,176.075,25.831,154.313
C06185=1082.809,317.759,410.577,176.079,25.838,154.314
C06186=1082.814,318.006,410.545,176.082,25.842,154.314
C06187=1082.820,318.254,410.513,176.085,25.846,154.315
C06188=1082.826,318.502,410.481,176.088,25.851,154.315
C06189=1082.832,318.750,410.447,176.091,25.855,154.316
C06190=1082.837,318.998,410.416,176.094,25.859,154.317
C06191=1082.844,319.245,410.383,176.097,25.863,154.317
C06192=1082.849,319.494,410.350,176.100,25.868,154.318
C06193=1082.855,319.741,410.318,176.103,25.872,154.319
C06194=1082.861,319.989,410.286,176.106,25.876,154.319
C06195=1082.867,320.236,410.253,176.109,25.880,154.320
C06196=1082.872,320.485,410.221,176.112,25.885,154.321
C06197=1082.878,320.733,410.188,176.115,25.889,154.321
C06198=1082.884,320.980,410.156,176.118,25.894,154.322
C06199=1082.889,321.228,410.123,176.121,25.897,154.322
C06200=1082.896,321.476,410.090,176.124,25.902,154.323
C06201=1082.902,321.724,410.058,176.127,25.906,154.324
C06202=1082.907,321.972,410.025,176.129,25.911,154.324
C06203=1082.913,322.219,409.993,176.132,25.915,154.325
C06204=1082.919,322.467,409.960,176.136,25.919,154.326
C06205=1082.924,322.715,409.927,176.138,25.923,154.326
C06206=1082.931,322.962,409.894,176.142,25.928,154.327
C06207=1082.937,323.211,409.862,176.145,25.932,154.327
C06208=1082.942,323.458,409.829,176.148,25.937,154.328
C06209=1082.949,323.706,409.796,176.151,25.941,154.329
C06210=1082.955,323.954,409.764,176.154,25.945,154.329
C06211=1082.959,324.201,409.731,176.157,25.949,154.330
C06212=1082.966,324.449,409.698,176.160,25.954,154.331
C06213=1082.972,324.697,409.666,176.163,25.958,154.331
C06214=1082.978,324.945,409.632,176.166,25.962,154.332
C06215=1082.984,325.193,409.600,176.169,25.967,154.333
C06216=1082.989,325.441,409.567,176.172,25.971,154.333
C06217=1082.995,325.688,409.534,176.175,25.976,154.334
C06218=1083.002,325.936,409.501,176.178,25.980,154.335
C06219=1083.007,326.184,409.468,176.181,25.984,154.335
C06220=1083.014,326.431,409.435,176.184,25.989,154.336
C06221=1083.019,326.679,409.402,176.187,25.993,154.337
C06222=1083.025,326.927,409.369,176.190,25.997,154.337
C06223=1083.031,327.175,409.336,176.194,26.002,154.338
C06224=1083.037,327.422,409.303,176.197,26.006,154.339
C06225=1083.044,327.670,409.270,176.200,26.011,154.339
C06226=1083.049,327.918,409.237,176.203,26.015,154.340
C06227=1083.055,328.165,409.204,176.206,26.020,154.341
C06228=1083.061,328.413,409.171,176.209,26.024,154.341
C06229=1083.067,328.661,409.138,176.212,26.028,154.342
C06230=1083.073,328.909,409.105,176.215,26.033,154.343
C06231=1083.079,329.156,409.072,176.217,26.037,154.343
C06232=1083.085,329.405,409.038,176.220,26.041,154.344
C06233=1083.092,329.653,409.006,176.223,26.046,154.344
C06234=1083.101,330.060,408.951,176.229,26.053,154.346
C06235=1083.111,330.469,408.896,176.234,26.061,154.347
C06236=1083.121,330.878,408.841,176.239,26.068,154.348
C06237=1083.131,331.286,408.786,176.244,26.075,154.349
C06238=1083.137,331.534,408.753,176.247,26.080,154.350
C06239=1083.143,331.781,408.720,176.250,26.084,154.350
C06240=1083.149,332.029,408.686,176.253,26.089,154.351
C06241=1083.154,332.277,408.653,176.256,26.093,154.352
C06242=1083.160,332.524,408.619,176.259,26.098,154.352
C06243=1083.167,332.772,408.586,176.262,26.102,154.353
C06244=1083.172,333.020,408.553,176.266,26.107,154.354
C06245=1083.179,333.268,408.518,176.269,26.111,154.354
C06246=1083.184,333.516,408.485,176.272,26.116,154.355
C06247=1083.190,333.764,408.452,176.275,26.121,154.356
C06248=1083.196,334.011,408.418,176.278,26.125,154.357
C06249=1083.202,334.259,408.385,176.281,26.130,154.357
C06250=1083.208,334.506,408.351,176.284,26.135,154.358
C06251=1083.213,334.754,408.317,176.287,26.139,154.359
C06252=1083.220,335.002,408.283,176.290,26.144,154.360
C06253=1083.225,335.250,408.250,176.293,26.149,154.360
C06254=1083.231,335.497,408.216,176.296,26.153,154.361
C06255=1083.238,335.744,408.183,176.299,26.158,154.362
C06256=1083.243,335.992,408.149,176.303,26.163,154.362
C06257=1083.250,336.240,408.115,176.306,26.167,154.363
C06258=1083.255,336.488,408.081,176.309,26.172,154.364
C06259=1083.261,336.735,408.047,176.312,26.176,154.365
C06260=1083.267,336.983,408.014,176.315,26.181,154.365
C06261=1083.273,337.230,407.980,176.318,26.186,154.366
C06262=1083.279,337.478,407.945,176.321,26.191,154.367
C06263=1083.285,337.726,407.912,176.324,26.195,154.367
C06264=1083.291,337.973,407.878,176.327,26.200,154.368
C06265=1083.298,338.221,407.844,176.330,26.205,154.369
C06266=1083.303,338.469,407.811,176.333,26.209,154.370
C06267=1083.308,338.716,407.776,176.337,26.214,154.370
C06268=1083.314,338.964,407.742,176.340,26.219,154.371
C06269=1083.321,339.212,407.708,176.343,26.224,154.372
C06270=1083.326,339.460,407.674,176.346,26.228,154.373
C06271=1083.332,339.707,407.640,176.350,26.233,154.373
C06272=1083.338,339.954,407.606,176.352,26.238,154.374
C06273=1083.344,340.202,407.572,176.355,26.243,154.375
C06274=1083.350,340.449,407.538,176.358,26.248,154.376
C06275=1083.356,340.697,407.504,176.361,26.252,154.376
C06276=1083.363,340.945,407.469,176.365,26.257,154.377
C06277=1083.368,341.192,407.435,176.368,26.262,154.378
C06278=1083.373,341.440,407.401,176.371,26.267,154.379
C06279=1083.380,341.688,407.367,176.374,26.272,154.380
C06280=1083.386,341.936,407.333,176.378,26.277,154.380
C06281=1083.392,342.183,407.299,176.380,26.282,154.381
C06282=1083.398,342.431,407.264,176.383,26.287,154.382
C06283=1083.404,342.678,407.230,176.386,26.292,154.383
C06284=1083.409,342.926,407.196,176.390,26.297,154.384
C06285=1083.416,343.173,407.160,176.393,26.301,154.384
C06286=1083.426,343.576,407.105,176.398,26.309,154.386
C06287=1083.435,343.979,407.049,176.403,26.317,154.387
C06288=1083.444,344.382,406.993,176.408,26.325,154.388
C06289=1083.455,344.784,406.937,176.414,26.333,154.389
C06290=1083.461,345.032,406.902,176.417,26.338,154.390
C06291=1083.466,345.280,406.868,176.419,26.343,154.391
C06292=1083.473,345.528,406.833,176.423,26.349,154.392
C06293=1083.479,345.774,406.799,176.426,26.353,154.393
C06294=1083.484,346.022,406.764,176.429,26.358,154.393
C06295=1083.490,346.270,406.729,176.433,26.363,154.394
C06296=1083.496,346.517,406.695,176.436,26.368,154.395
C06297=1083.502,346.765,406.660,176.438,26.373,154.396
C06298=1083.508,347.012,406.626,176.441,26.378,154.397
C06299=1083.514,347.260,406.591,176.445,26.383,154.397
C06300=1083.520,347.507,406.556,176.448,26.389,154.398
C06301=1083.526,347.755,406.521,176.451,26.393,154.399
C06302=1083.532,348.002,406.486,176.455,26.399,154.400
C06303=1083.538,348.250,406.452,176.458,26.404,154.401
C06304=1083.544,348.497,406.416,176.460,26.409,154.402
C06305=1083.550,348.745,406.382,176.464,26.414,154.402
C06306=1083.555,348.993,406.347,176.467,26.419,154.403
C06307=1083.562,349.240,406.312,176.470,26.424,154.404
C06308=1083.567,349.488,406.277,176.474,26.430,154.405
C06309=1083.574,349.735,406.242,176.477,26.434,154.406
C06310=1083.579,349.982,406.207,176.479,26.440,154.407
C06311=1083.586,350.230,406.173,176.483,26.445,154.408
C06312=1083.591,350.477,406.137,176.486,26.450,154.408
C06313=1083.598,350.725,406.103,176.489,26.455,154.409
C06314=1083.604,350.973,406.067,176.493,26.460,154.410
C06315=1083.610,351.219,406.032,176.496,26.465,154.411
C06316=1083.616,351.468,405.997,176.499,26.471,154.412
C06317=1083.622,351.714,405.962,176.502,26.476,154.413
C06318=1083.628,351.962,405.927,176.505,26.481,154.414
C06319=1083.634,352.210,405.892,176.509,26.487,154.414
C06320=1083.640,352.457,405.857,176.512,26.491,154.415
C06321=1083.646,352.704,405.821,176.515,26.497,154.416
C06322=1083.653,352.952,405.786,176.518,26.502,154.417
C06323=1083.658,353.199,405.751,176.521,26.507,154.418
C06324=1083.664,353.447,405.716,176.525,26.513,154.419
C06325=1083.670,353.694,405.681,176.528,26.518,154.420
C06326=1083.676,353.941,405.645,176.531,26.523,154.421
C06327=1083.682,354.189,405.609,176.534,26.529,154.422
C06328=1083.688,354.436,405.575,176.537,26.534,154.422
C06329=1083.694,354.683,405.539,176.541,26.539,154.423
C06330=1083.700,354.931,405.503,176.544,26.544,154.424
C06331=1083.705,355.179,405.469,176.547,26.550,154.425
C06332=1083.711,355.426,405.433,176.550,26.555,154.426
C06333=1083.718,355.674,405.398,176.553,26.561,154.427
C06334=1083.724,355.921,405.362,176.557,26.566,154.428
C06335=1083.730,356.168,405.327,176.560,26.571,154.429
C06336=1083.736,356.416,405.291,176.563,26.577,154.430
C06337=1083.743,356.663,405.255,176.566,26.582,154.431
C06338=1083.752,357.069,405.197,176.572,26.591,154.432
C06339=1083.762,357.474,405.139,176.576,26.600,154.434
C06340=1083.772,357.880,405.080,176.582,26.609,154.435
C06341=1083.781,358.286,405.022,176.588,26.618,154.437
C06342=1083.788,358.533,404.986,176.590,26.623,154.438
C06343=1083.794,358.781,404.950,176.594,26.629,154.438
C06344=1083.800,359.028,404.914,176.597,26.635,154.440
C06345=1083.806,359.275,404.879,176.601,26.640,154.440
C06346=1083.812,359.522,404.843,176.603,26.645,154.441
C06347=1083.818,359.770,404.807,176.607,26.651,154.442
C06348=1083.824,360.018,404.771,176.610,26.657,154.443
C06349=1083.830,360.265,404.735,176.614,26.662,154.444
C06350=1083.836,360.512,404.699,176.617,26.668,154.445
C06351=1083.842,360.759,404.664,176.620,26.674,154.446
C06352=1083.848,361.006,404.627,176.623,26.679,154.447
C06353=1083.854,361.254,404.591,176.627,26.685,154.448
C06354=1083.861,361.501,404.555,176.630,26.690,154.449
C06355=1083.867,361.749,404.519,176.633,26.696,154.450
C06356=1083.873,361.997,404.484,176.636,26.702,154.451
C06357=1083.878,362.243,404.447,176.640,26.708,154.452
C06358=1083.884,362.491,404.412,176.643,26.713,154.453
C06359=1083.891,362.738,404.375,176.646,26.719,154.454
C06360=1083.897,362.985,404.339,176.649,26.724,154.455
C06361=1083.903,363.232,404.303,176.653,26.730,154.456
C06362=1083.909,363.479,404.267,176.656,26.736,154.457
C06363=1083.915,363.727,404.231,176.659,26.742,154.458
C06364=1083.922,363.974,404.195,176.662,26.747,154.459
C06365=1083.928,364.222,404.159,176.666,26.753,154.460
C06366=1083.933,364.469,404.122,176.669,26.759,154.461
C06367=1083.940,364.716,404.085,176.672,26.765,154.462
C06368=1083.945,364.963,404.049,176.675,26.770,154.463
C06369=1083.952,365.210,404.014,176.679,26.776,154.464
C06370=1083.958,365.457,403.977,176.682,26.782,154.465
C06371=1083.964,365.704,403.941,176.685,26.788,154.466
C06372=1083.970,365.952,403.904,176.689,26.794,154.467
C06373=1083.976,366.199,403.868,176.692,26.799,154.468
C06374=1083.982,366.446,403.831,176.695,26.806,154.469
C06375=1083.988,366.694,403.794,176.698,26.811,154.470
C06376=1083.994,366.941,403.758,176.702,26.817,154.471
C06377=1084.000,367.188,403.721,176.705,26.824,154.472
C06378=1084.006,367.435,403.684,176.708,26.830,154.473
C06379=1084.012,367.682,403.648,176.711,26.835,154.474
C06380=1084.018,367.930,403.612,176.715,26.841,154.475
C06381=1084.024,368.177,403.575,176.718,26.847,154.476
C06382=1084.030,368.424,403.539,176.721,26.853,154.478
C06383=1084.037,368.672,403.502,176.725,26.859,154.479
C06384=1084.042,368.919,403.465,176.728,26.865,154.480
C06385=1084.049,369.166,403.429,176.731,26.871,154.481
C06386=1084.055,369.412,403.392,176.735,26.877,154.482
C06387=1084.061,369.660,403.355,176.738,26.883,154.483
C06388=1084.067,369.907,403.318,176.741,26.890,154.484
C06389=1084.073,370.154,403.281,176.744,26.895,154.485
C06390=1084.079,370.365,403.250,176.747,26.901,154.486
C06391=1084.084,370.576,403.219,176.750,26.906,154.487
C06392=1084.088,370.787,403.187,176.753,26.911,154.488
C06393=1084.094,370.998,403.156,176.756,26.916,154.489
C06394=1084.100,371.208,403.124,176.759,26.921,154.490
C06395=1084.105,371.419,403.092,176.761,26.927,154.491
C06396=1084.110,371.629,403.061,176.764,26.932,154.492
C06397=1084.115,371.841,403.030,176.767,26.937,154.493
C06398=1084.121,372.088,402.993,176.771,26.944,154.494
C06399=1084.127,372.335,402.956,176.774,26.949,154.495
C06400=1084.134,372.583,402.919,176.777,26.956,154.496
C06401=1084.140,372.829,402.881,176.780,26.962,154.497
C06402=1084.146,373.077,402.845,176.784,26.968,154.498
C06403=1084.153,373.324,402.808,176.787,26.974,154.499
C06404=1084.158,373.570,402.771,176.790,26.980,154.500
C06405=1084.165,373.818,402.734,176.794,26.987,154.501
C06406=1084.171,374.065,402.696,176.797,26.993,154.503
C06407=1084.177,374.312,402.659,176.800,26.999,154.504
C06408=1084.183,374.559,402.623,176.804,27.006,154.505
C06409=1084.189,374.806,402.585,176.807,27.012,154.506
C06410=1084.195,375.053,402.548,176.810,27.018,154.507
C06411=1084.201,375.301,402.510,176.814,27.025,154.508
C06412=1084.208,375.547,402.472,176.817,27.031,154.510
C06413=1084.213,375.795,402.435,176.820,27.038,154.511
C06414=1084.219,376.041,402.398,176.824,27.044,154.512
C06415=1084.226,376.288,402.361,176.827,27.051,154.513
C06416=1084.232,376.536,402.323,176.831,27.057,154.514
C06417=1084.238,376.783,402.285,176.834,27.063,154.516
C06418=1084.244,377.030,402.248,176.837,27.070,154.517
C06419=1084.250,377.276,402.211,176.841,27.077,154.518
C06420=1084.257,377.524,402.173,176.843,27.083,154.519
C06421=1084.263,377.771,402.135,176.847,27.089,154.520
C06422=1084.268,378.018,402.098,176.851,27.096,154.521
C06423=1084.276,378.265,402.061,176.854,27.103,154.523
C06424=1084.282,378.512,402.023,176.857,27.109,154.524
C06425=1084.287,378.759,401.985,176.861,27.115,154.525
C06426=1084.294,379.006,401.947,176.864,27.122,154.526
C06427=1084.300,379.253,401.910,176.868,27.129,154.528
C06428=1084.306,379.500,401.873,176.871,27.135,154.529
C06429=1084.313,379.747,401.835,176.874,27.142,154.530
C06430=1084.319,379.994,401.797,176.878,27.149,154.531
C06431=1084.324,380.241,401.759,176.881,27.155,154.532
C06432=1084.331,380.488,401.721,176.884,27.162,154.534
C06433=1084.337,380.735,401.683,176.888,27.168,154.535
C06434=1084.344,380.982,401.646,176.891,27.175,154.536
C06435=1084.350,381.229,401.608,176.895,27.182,154.537
C06436=1084.356,381.476,401.570,176.898,27.189,154.539
C06437=1084.362,381.723,401.532,176.901,27.195,154.540
C06438=1084.368,381.970,401.494,176.905,27.202,154.541
C06439=1084.375,382.217,401.456,176.908,27.209,154.542
C06440=1084.381,382.463,401.418,176.912,27.216,154.544
C06441=1084.388,382.711,401.380,176.915,27.222,154.545
C06442=1084.393,382.957,401.342,176.918,27.229,154.546
C06443=1084.399,383.204,401.304,176.922,27.236,154.548
C06444=1084.406,383.452,401.266,176.925,27.243,154.549
C06445=1084.412,383.698,401.228,176.929,27.250,154.550
C06446=1084.417,383.923,401.193,176.932,27.257,154.552
C06447=1084.424,384.148,401.158,176.934,27.263,154.553
C06448=1084.429,384.373,401.123,176.938,27.269,154.554
C06449=1084.435,384.597,401.089,176.941,27.276,154.555
C06450=1084.440,384.823,401.054,176.945,27.282,154.556
C06451=1084.446,385.048,401.018,176.947,27.289,154.558
C06452=1084.452,385.273,400.984,176.951,27.295,154.559
C06453=1084.457,385.497,400.949,176.954,27.301,154.560
C06454=1084.463,385.745,400.911,176.957,27.309,154.561
C06455=1084.470,385.991,400.872,176.961,27.315,154.563
C06456=1084.476,386.238,400.834,176.964,27.322,154.564
C06457=1084.482,386.485,400.796,176.967,27.330,154.565
C06458=1084.488,386.732,400.757,176.971,27.336,154.567
C06459=1084.494,386.978,400.718,176.974,27.344,154.568
C06460=1084.501,387.226,400.680,176.978,27.351,154.569
C06461=1084.508,387.473,400.641,176.981,27.358,154.571
C06462=1084.514,387.719,400.604,176.985,27.366,154.572
C06463=1084.520,387.967,400.564,176.988,27.372,154.573
C06464=1084.526,388.213,400.526,176.992,27.380,154.575
C06465=1084.532,388.460,400.488,176.995,27.387,154.576
C06466=1084.539,388.707,400.449,176.998,27.394,154.578
C06467=1084.545,388.953,400.410,177.002,27.401,154.579
C06468=1084.551,389.201,400.372,177.005,27.409,154.580
C06469=1084.558,389.448,400.333,177.009,27.416,154.582
C06470=1084.564,389.694,400.294,177.012,27.423,154.583
C06471=1084.571,389.941,400.256,177.016,27.430,154.585
C06472=1084.576,390.187,400.216,177.019,27.438,154.586
C06473=1084.583,390.435,400.178,177.023,27.445,154.587
C06474=1084.590,390.681,400.139,177.026,27.452,154.589
C06475=1084.596,390.928,400.100,177.030,27.460,154.590
C06476=1084.602,391.175,400.062,177.033,27.467,154.592
C06477=1084.609,391.421,400.023,177.037,27.475,154.593
C06478=1084.615,391.669,399.983,177.040,27.482,154.595
C06479=1084.622,391.915,399.944,177.044,27.490,154.596
C06480=1084.628,392.162,399.906,177.048,27.497,154.598
C06481=1084.634,392.409,399.867,177.051,27.505,154.599
C06482=1084.641,392.655,399.828,177.055,27.512,154.600
C06483=1084.647,392.903,399.788,177.058,27.520,154.602
C06484=1084.653,393.149,399.750,177.062,27.528,154.603
C06485=1084.659,393.396,399.710,177.065,27.535,154.605
C06486=1084.666,393.643,399.672,177.069,27.543,154.606
C06487=1084.672,393.890,399.632,177.072,27.551,154.608
C06488=1084.678,394.137,399.593,177.076,27.558,154.609
C06489=1084.685,394.383,399.553,177.079,27.566,154.611
C06490=1084.691,394.630,399.514,177.083,27.574,154.612
C06491=1084.698,394.876,399.475,177.086,27.581,154.614
C06492=1084.704,395.124,399.436,177.090,27.589,154.615
C06493=1084.710,395.370,399.396,177.093,27.597,154.617
C06494=1084.717,395.617,399.357,177.097,27.605,154.619
C06495=1084.723,395.864,399.317,177.100,27.612,154.620
C06496=1084.729,396.111,399.278,177.104,27.620,154.622
C06497=1084.735,396.357,399.239,177.107,27.628,154.623
C06498=1084.742,396.604,399.199,177.111,27.636,154.625
C06499=1084.748,396.850,399.159,177.114,27.644,154.626
C06500=1084.755,397.097,399.120,177.118,27.652,154.628
C06501=1084.761,397.344,399.081,177.121,27.660,154.629
C06502=1084.767,397.575,399.043,177.125,27.667,154.631
C06503=1084.773,397.807,399.006,177.128,27.675,154.632
C06504=1084.779,398.038,398.969,177.131,27.682,154.634
C06505=1084.785,398.270,398.932,177.134,27.690,154.635
C06506=1084.791,398.502,398.895,177.138,27.697,154.637
C06507=1084.797,398.733,398.857,177.141,27.705,154.638
C06508=1084.803,398.964,398.820,177.145,27.712,154.640
C06509=1084.809,399.196,398.783,177.148,27.720,154.641
C06510=1084.815,399.444,398.743,177.151,27.728,154.643
C06511=1084.821,399.691,398.703,177.155,27.737,154.645
C06512=1084.828,399.938,398.663,177.159,27.745,154.646
C06513=1084.835,400.186,398.623,177.162,27.753,154.648
C06514=1084.841,400.433,398.583,177.166,27.761,154.650
C06515=1084.848,400.679,398.543,177.169,27.769,154.651
C06516=1084.854,400.926,398.503,177.173,27.778,154.653
C06517=1084.860,401.173,398.463,177.176,27.786,154.655
C06518=1084.866,401.419,398.423,177.181,27.795,154.656
C06519=1084.873,401.666,398.383,177.184,27.803,154.658
C06520=1084.879,401.912,398.343,177.187,27.811,154.660
C06521=1084.886,402.159,398.303,177.191,27.819,154.661
C06522=1084.893,402.406,398.262,177.194,27.828,154.663
C06523=1084.899,402.653,398.222,177.198,27.836,154.665
C06524=1084.905,402.899,398.182,177.202,27.845,154.667
C06525=1084.912,403.146,398.142,177.206,27.853,154.668
C06526=1084.918,403.392,398.102,177.209,27.862,154.670
C06527=1084.925,403.639,398.061,177.213,27.870,154.672
C06528=1084.931,403.886,398.021,177.217,27.879,154.673
C06529=1084.938,404.133,397.981,177.220,27.887,154.675
C06530=1084.944,404.379,397.941,177.224,27.896,154.677
C06531=1084.951,404.626,397.900,177.227,27.905,154.679
C06532=1084.958,404.873,397.860,177.232,27.913,154.680
C06533=1084.964,405.119,397.820,177.235,27.922,154.682
C06534=1084.970,405.366,397.779,177.238,27.931,154.684
C06535=1084.976,405.612,397.738,177.242,27.939,154.686
C06536=1084.983,405.859,397.698,177.246,27.948,154.687
C06537=1084.990,406.106,397.657,177.250,27.957,154.689
C06538=1084.996,406.352,397.617,177.253,27.966,154.691
C06539=1085.002,406.598,397.576,177.256,27.974,154.693
C06540=1085.009,406.846,397.535,177.261,27.984,154.695
C06541=1085.015,407.092,397.495,177.264,27.992,154.696
C06542=1085.022,407.338,397.454,177.268,28.001,154.698
C06543=1085.028,407.586,397.413,177.272,28.010,154.700
C06544=1085.035,407.831,397.372,177.275,28.019,154.702
C06545=1085.041,408.078,397.332,177.279,28.028,154.704
C06546=1085.048,408.325,397.290,177.283,28.037,154.706
C06547=1085.054,408.571,397.250,177.287,28.046,154.707
C06548=1085.060,408.818,397.209,177.291,28.056,154.709
C06549=1085.067,409.065,397.168,177.294,28.065,154.711
C06550=1085.073,409.311,397.127,177.298,28.073,154.713
C06551=1085.080,409.558,397.086,177.302,28.083,154.715
C06552=1085.087,409.804,397.045,177.305,28.092,154.717
C06553=1085.093,410.050,397.004,177.309,28.101,154.719
C06554=1085.100,410.298,396.963,177.313,28.111,154.721
C06555=1085.106,410.544,396.922,177.317,28.119,154.723
C06556=1085.113,410.790,396.881,177.321,28.129,154.725
C06557=1085.119,411.037,396.839,177.324,28.139,154.727
C06558=1085.125,411.270,396.801,177.328,28.147,154.728
C06559=1085.131,411.502,396.762,177.331,28.156,154.730
C06560=1085.138,411.735,396.723,177.336,28.165,154.732
C06561=1085.144,411.968,396.684,177.339,28.174,154.734
C06562=1085.150,412.200,396.645,177.342,28.183,154.736
C06563=1085.156,412.433,396.606,177.346,28.191,154.738
C06564=1085.162,412.665,396.567,177.349,28.201,154.739
C06565=1085.169,412.898,396.528,177.353,28.209,154.741
C06566=1085.175,413.145,396.486,177.357,28.219,154.743
C06567=1085.182,413.391,396.445,177.361,28.228,154.745
C06568=1085.189,413.638,396.404,177.365,28.238,154.747
C06569=1085.195,413.884,396.363,177.369,28.248,154.749
C06570=1085.202,414.131,396.321,177.373,28.257,154.751
C06571=1085.209,414.377,396.280,177.377,28.267,154.753
C06572=1085.215,414.623,396.238,177.380,28.277,154.755
C06573=1085.222,414.870,396.197,177.385,28.287,154.757
C06574=1085.229,415.116,396.154,177.388,28.296,154.759
C06575=1085.235,415.362,396.113,177.392,28.306,154.762
C06576=1085.242,415.609,396.072,177.396,28.316,154.764
C06577=1085.249,415.856,396.030,177.400,28.326,154.766
C06578=1085.255,416.102,395.988,177.404,28.336,154.768
C06579=1085.263,416.348,395.946,177.408,28.346,154.770
C06580=1085.269,416.595,395.905,177.412,28.356,154.772
C06581=1085.275,416.841,395.862,177.416,28.366,154.774
C06582=1085.282,417.088,395.821,177.420,28.376,154.776
C06583=1085.288,417.334,395.779,177.424,28.386,154.778
C06584=1085.295,417.580,395.737,177.427,28.396,154.780
C06585=1085.302,417.827,395.695,177.431,28.406,154.783
C06586=1085.309,418.073,395.653,177.436,28.416,154.785
C06587=1085.316,418.319,395.610,177.439,28.426,154.787
C06588=1085.322,418.565,395.569,177.443,28.437,154.789
C06589=1085.329,418.812,395.526,177.448,28.447,154.791
C06590=1085.335,419.059,395.485,177.452,28.457,154.793
C06591=1085.342,419.305,395.442,177.455,28.467,154.796
C06592=1085.348,419.550,395.400,177.460,28.478,154.798
C06593=1085.355,419.797,395.358,177.464,28.488,154.800
C06594=1085.362,420.044,395.315,177.467,28.499,154.802
C06595=1085.369,420.290,395.273,177.471,28.509,154.804
C06596=1085.376,420.536,395.231,177.476,28.520,154.807
C06597=1085.383,420.782,395.188,177.480,28.530,154.809
C06598=1085.389,421.029,395.147,177.483,28.541,154.811
C06599=1085.396,421.275,395.104,177.488,28.551,154.813
C06600=1085.403,421.521,395.062,177.492,28.562,154.816
C06601=1085.409,421.767,395.019,177.496,28.572,154.818
C06602=1085.416,422.014,394.977,177.501,28.583,154.820
C06603=1085.423,422.260,394.934,177.504,28.593,154.822
C06604=1085.430,422.506,394.892,177.508,28.604,154.825
C06605=1085.436,422.753,394.849,177.512,28.615,154.827
C06606=1085.443,422.999,394.806,177.517,28.626,154.829
C06607=1085.450,423.245,394.764,177.521,28.637,154.832
C06608=1085.457,423.492,394.721,177.525,28.648,154.834
C06609=1085.464,423.737,394.678,177.528,28.659,154.836
C06610=1085.471,423.983,394.635,177.533,28.669,154.839
C06611=1085.477,424.230,394.592,177.537,28.681,154.841
C06612=1085.484,424.476,394.550,177.541,28.692,154.844
C06613=1085.491,424.722,394.506,177.546,28.703,154.846
C06614=1085.497,424.962,394.465,177.550,28.714,154.848
C06615=1085.504,425.203,394.423,177.554,28.725,154.851
C06616=1085.510,425.443,394.381,177.557,28.736,154.853
C06617=1085.517,425.684,394.339,177.562,28.746,154.855
C06618=1085.524,425.925,394.297,177.566,28.758,154.858
C06619=1085.530,426.165,394.254,177.570,28.768,154.860
C06620=1085.537,426.406,394.212,177.575,28.779,154.863
C06621=1085.544,426.647,394.170,177.578,28.790,154.865
C06622=1085.551,426.893,394.127,177.582,28.802,154.867
C06623=1085.557,427.139,394.084,177.586,28.813,154.870
C06624=1085.565,427.385,394.041,177.591,28.825,154.872
C06625=1085.572,427.630,393.998,177.595,28.836,154.875
C06626=1085.578,427.877,393.954,177.599,28.847,154.877
C06627=1085.586,428.123,393.911,177.604,28.859,154.880
C06628=1085.592,428.369,393.867,177.608,28.871,154.882
C06629=1085.599,428.615,393.824,177.612,28.882,154.885
C06630=1085.606,428.861,393.781,177.616,28.894,154.888
C06631=1085.613,429.107,393.737,177.621,28.906,154.890
C06632=1085.620,429.353,393.694,177.626,28.918,154.893
C06633=1085.627,429.599,393.650,177.630,28.929,154.895
C06634=1085.634,429.845,393.607,177.634,28.941,154.898
C06635=1085.640,430.091,393.563,177.639,28.953,154.900
C06636=1085.647,430.337,393.519,177.643,28.965,154.903
C06637=1085.655,430.583,393.475,177.647,28.977,154.906
C06638=1085.661,430.829,393.431,177.651,28.989,154.908
C06639=1085.668,431.075,393.388,177.655,29.001,154.911
C06640=1085.675,431.322,393.344,177.660,29.013,154.914
C06641=1085.682,431.567,393.301,177.664,29.025,154.916
C06642=1085.689,431.813,393.257,177.669,29.037,154.919
C06643=1085.696,432.060,393.213,177.674,29.049,154.922
C06644=1085.703,432.305,393.169,177.678,29.062,154.924
C06645=1085.710,432.551,393.125,177.682,29.074,154.927
C06646=1085.717,432.797,393.081,177.686,29.086,154.930
C06647=1085.724,433.043,393.037,177.691,29.099,154.933
C06648=1085.731,433.289,392.993,177.696,29.111,154.935
C06649=1085.738,433.535,392.948,177.700,29.124,154.938
C06650=1085.744,433.781,392.904,177.704,29.136,154.941
C06651=1085.751,434.026,392.861,177.708,29.149,154.944
C06652=1085.759,434.272,392.816,177.714,29.161,154.947
C06653=1085.765,434.518,392.772,177.718,29.174,154.949
C06654=1085.773,434.765,392.727,177.722,29.187,154.952
C06655=1085.779,435.011,392.683,177.726,29.199,154.955
C06656=1085.786,435.257,392.638,177.732,29.212,154.958
C06657=1085.794,435.502,392.594,177.736,29.225,154.961
C06658=1085.801,435.748,392.550,177.740,29.237,154.963
C06659=1085.808,435.994,392.505,177.745,29.251,154.966
C06660=1085.815,436.240,392.460,177.749,29.264,154.969
C06661=1085.822,436.485,392.416,177.754,29.277,154.972
C06662=1085.829,436.732,392.372,177.759,29.289,154.975
C06663=1085.835,436.977,392.327,177.763,29.302,154.978
C06664=1085.843,437.223,392.282,177.767,29.315,154.981
C06665=1085.849,437.468,392.238,177.773,29.329,154.984
C06666=1085.857,437.714,392.193,177.777,29.342,154.987
C06667=1085.865,437.960,392.148,177.781,29.355,154.990
C06668=1085.872,438.206,392.104,177.786,29.368,154.993
C06669=1085.879,438.452,392.059,177.791,29.382,154.996
C06670=1085.885,438.667,392.019,177.795,29.394,154.999
C06671=1085.891,438.884,391.980,177.800,29.405,155.001
C06672=1085.898,439.100,391.940,177.803,29.417,155.004
C06673=1085.903,439.316,391.901,177.807,29.429,155.006
C06674=1085.910,439.533,391.861,177.812,29.441,155.009
C06675=1085.917,439.749,391.821,177.815,29.453,155.012
C06676=1085.923,439.965,391.782,177.820,29.465,155.015
C06677=1085.929,440.181,391.742,177.824,29.477,155.017
C06678=1085.937,440.427,391.697,177.829,29.491,155.020
C06679=1085.944,440.673,391.651,177.834,29.504,155.023
C06680=1085.951,440.919,391.606,177.838,29.518,155.027
C06681=1085.958,441.164,391.562,177.843,29.532,155.030
C06682=1085.965,441.409,391.516,177.848,29.546,155.033
C06683=1085.973,441.655,391.471,177.853,29.560,155.036
C06684=1085.979,441.901,391.425,177.857,29.574,155.039
C06685=1085.987,442.147,391.380,177.862,29.588,155.042
C06686=1085.994,442.392,391.335,177.867,29.602,155.046
C06687=1086.001,442.637,391.289,177.872,29.616,155.049
C06688=1086.008,442.884,391.243,177.877,29.631,155.052
C06689=1086.016,443.129,391.198,177.881,29.645,155.055
C06690=1086.023,443.375,391.152,177.887,29.659,155.059
C06691=1086.030,443.620,391.106,177.891,29.673,155.062
C06692=1086.038,443.866,391.060,177.896,29.688,155.065
C06693=1086.045,444.112,391.015,177.901,29.703,155.069
C06694=1086.052,444.357,390.969,177.906,29.717,155.072
C06695=1086.059,444.602,390.924,177.911,29.731,155.075
C06696=1086.067,444.848,390.878,177.916,29.746,155.079
C06697=1086.074,445.094,390.832,177.920,29.761,155.082
C06698=1086.081,445.339,390.786,177.926,29.776,155.086
C06699=1086.088,445.585,390.740,177.930,29.790,155.089
C06700=1086.096,445.830,390.694,177.934,29.805,155.092
C06701=1086.103,446.075,390.647,177.939,29.819,155.096
C06702=1086.111,446.321,390.602,177.942,29.834,155.099
C06703=1086.118,446.567,390.555,177.945,29.849,155.103
C06704=1086.126,446.813,390.510,177.949,29.863,155.106
C06705=1086.133,447.058,390.463,177.952,29.878,155.110
C06706=1086.140,447.303,390.416,177.955,29.892,155.113
C06707=1086.148,447.549,390.371,177.958,29.907,155.117
C06708=1086.155,447.795,390.324,177.960,29.921,155.120
C06709=1086.162,448.039,390.278,177.962,29.936,155.124
C06710=1086.169,448.285,390.232,177.965,29.951,155.127
C06711=1086.178,448.531,390.186,177.967,29.966,155.131
C06712=1086.185,448.776,390.139,177.969,29.980,155.134
C06713=1086.192,449.022,390.093,177.971,29.994,155.138
C06714=1086.200,449.267,390.046,177.973,30.009,155.142
C06715=1086.208,449.512,390.000,177.974,30.023,155.145
C06716=1086.217,449.758,389.954,177.975,30.037,155.149
C06717=1086.228,450.004,389.910,177.976,30.050,155.152
C06718=1085.852,449.996,389.706,177.941,30.235,155.202
C06719=1085.841,449.749,389.751,177.939,30.222,155.199
C06720=1085.831,449.504,389.798,177.938,30.208,155.195
C06721=1085.823,449.259,389.844,177.936,30.194,155.192
C06722=1085.817,449.015,389.890,177.935,30.179,155.188
C06723=1085.808,448.768,389.937,177.933,30.165,155.184
C06724=1085.801,448.523,389.983,177.930,30.150,155.181
C06725=1085.794,448.278,390.029,177.928,30.136,155.177
C06726=1085.786,448.033,390.076,177.926,30.121,155.174
C06727=1085.779,447.786,390.123,177.924,30.106,155.170
C06728=1085.771,447.541,390.168,177.920,30.092,155.167
C06729=1085.764,447.296,390.215,177.918,30.077,155.163
C06730=1085.756,447.050,390.261,177.914,30.063,155.160
C06731=1085.749,446.805,390.308,177.911,30.048,155.156
C06732=1085.742,446.559,390.354,177.908,30.033,155.153
C06733=1085.735,446.314,390.400,177.904,30.019,155.149
C06734=1085.728,446.068,390.446,177.901,30.004,155.146
C06735=1085.719,445.823,390.493,177.896,29.990,155.142
C06736=1085.712,445.577,390.539,177.892,29.975,155.139
C06737=1085.705,445.332,390.585,177.887,29.960,155.135
C06738=1085.698,445.086,390.631,177.882,29.945,155.132
C06739=1085.690,444.840,390.677,177.878,29.930,155.128
C06740=1085.683,444.595,390.722,177.872,29.916,155.125
C06741=1085.676,444.349,390.768,177.867,29.901,155.122
C06742=1085.668,444.104,390.814,177.863,29.887,155.118
C06743=1085.661,443.858,390.860,177.857,29.872,155.115
C06744=1085.653,443.613,390.906,177.852,29.857,155.112
C06745=1085.646,443.367,390.952,177.848,29.843,155.108
C06746=1085.640,443.122,390.997,177.842,29.829,155.105
C06747=1085.632,442.877,391.043,177.837,29.815,155.102
C06748=1085.625,442.631,391.088,177.832,29.800,155.099
C06749=1085.618,442.385,391.134,177.827,29.786,155.095
C06750=1085.610,442.139,391.180,177.823,29.772,155.092
C06751=1085.603,441.893,391.225,177.817,29.758,155.089
C06752=1085.595,441.648,391.271,177.813,29.744,155.086
C06753=1085.588,441.402,391.317,177.808,29.730,155.083
C06754=1085.581,441.157,391.361,177.803,29.716,155.079
C06755=1085.574,440.911,391.407,177.798,29.702,155.076
C06756=1085.566,440.665,391.452,177.794,29.688,155.073
C06757=1085.559,440.419,391.497,177.788,29.674,155.070
C06758=1085.551,440.174,391.542,177.784,29.661,155.067
C06759=1085.546,439.965,391.581,177.779,29.649,155.064
C06760=1085.540,439.756,391.619,177.776,29.637,155.061
C06761=1085.534,439.547,391.657,177.771,29.626,155.059
C06762=1085.528,439.338,391.697,177.768,29.614,155.056
C06763=1085.522,439.129,391.735,177.763,29.603,155.054
C06764=1085.515,438.920,391.773,177.760,29.591,155.051
C06765=1085.509,438.711,391.811,177.755,29.580,155.049
C06766=1085.502,438.502,391.849,177.751,29.568,155.046
C06767=1085.496,438.256,391.893,177.746,29.555,155.043
C06768=1085.488,438.010,391.938,177.742,29.542,155.040
C06769=1085.481,437.764,391.983,177.737,29.529,155.037
C06770=1085.474,437.519,392.028,177.732,29.516,155.034
C06771=1085.467,437.273,392.073,177.728,29.502,155.031
C06772=1085.460,437.027,392.118,177.722,29.489,155.028
C06773=1085.453,436.781,392.162,177.718,29.476,155.025
C06774=1085.446,436.535,392.207,177.714,29.463,155.022
C06775=1085.439,436.290,392.252,177.709,29.450,155.019
C06776=1085.431,436.044,392.297,177.704,29.437,155.016
C06777=1085.424,435.798,392.342,177.700,29.424,155.014
C06778=1085.417,435.552,392.385,177.695,29.411,155.011
C06779=1085.410,435.306,392.430,177.690,29.398,155.008
C06780=1085.403,435.061,392.474,177.686,29.385,155.005
C06781=1085.396,434.814,392.519,177.681,29.373,155.002
C06782=1085.389,434.569,392.563,177.677,29.360,154.999
C06783=1085.382,434.323,392.608,177.672,29.347,154.996
C06784=1085.375,434.077,392.652,177.667,29.335,154.994
C06785=1085.368,433.832,392.696,177.663,29.322,154.991
C06786=1085.361,433.585,392.740,177.659,29.310,154.988
C06787=1085.354,433.340,392.785,177.653,29.297,154.985
C06788=1085.347,433.093,392.829,177.649,29.285,154.983
C06789=1085.340,432.848,392.874,177.645,29.272,154.980
C06790=1085.333,432.602,392.917,177.641,29.260,154.977
C06791=1085.326,432.355,392.961,177.636,29.247,154.974
C06792=1085.320,432.110,393.006,177.632,29.235,154.972
C06793=1085.312,431.864,393.049,177.627,29.223,154.969
C06794=1085.305,431.618,393.093,177.622,29.211,154.966
C06795=1085.298,431.372,393.136,177.618,29.199,154.964
C06796=1085.291,431.126,393.181,177.614,29.187,154.961
C06797=1085.284,430.880,393.225,177.609,29.175,154.958
C06798=1085.277,430.634,393.268,177.605,29.163,154.955
C06799=1085.271,430.388,393.312,177.601,29.151,154.953
C06800=1085.263,430.142,393.356,177.596,29.139,154.950
C06801=1085.257,429.896,393.400,177.592,29.127,154.948
C06802=1085.249,429.650,393.443,177.587,29.115,154.945
C06803=1085.242,429.404,393.487,177.582,29.103,154.942
C06804=1085.235,429.158,393.530,177.578,29.091,154.940
C06805=1085.229,428.912,393.574,177.574,29.079,154.937
C06806=1085.222,428.666,393.617,177.569,29.068,154.935
C06807=1085.215,428.420,393.661,177.565,29.056,154.932
C06808=1085.208,428.173,393.704,177.561,29.044,154.930
C06809=1085.201,427.927,393.748,177.556,29.033,154.927
C06810=1085.194,427.682,393.791,177.552,29.021,154.924
C06811=1085.187,427.435,393.834,177.548,29.010,154.922
C06812=1085.180,427.189,393.878,177.543,28.998,154.920
C06813=1085.173,426.943,393.921,177.539,28.987,154.917
C06814=1085.166,426.697,393.964,177.535,28.975,154.915
C06815=1085.159,426.456,394.006,177.531,28.964,154.912
C06816=1085.153,426.215,394.049,177.527,28.953,154.910
C06817=1085.146,425.974,394.091,177.522,28.943,154.907
C06818=1085.139,425.732,394.133,177.518,28.931,154.905
C06819=1085.133,425.491,394.176,177.514,28.920,154.903
C06820=1085.126,425.250,394.218,177.509,28.909,154.900
C06821=1085.119,425.009,394.260,177.506,28.898,154.898
C06822=1085.112,424.768,394.302,177.502,28.888,154.895
C06823=1085.106,424.521,394.345,177.497,28.876,154.893
C06824=1085.099,424.276,394.388,177.493,28.865,154.891
C06825=1085.092,424.030,394.431,177.489,28.854,154.888
C06826=1085.085,423.783,394.473,177.484,28.843,154.886
C06827=1085.079,423.537,394.516,177.481,28.832,154.883
C06828=1085.072,423.291,394.560,177.477,28.822,154.881
C06829=1085.065,423.045,394.602,177.472,28.810,154.879
C06830=1085.058,422.798,394.645,177.468,28.800,154.876
C06831=1085.051,422.552,394.687,177.464,28.789,154.874
C06832=1085.045,422.306,394.730,177.459,28.778,154.872
C06833=1085.039,422.059,394.773,177.456,28.768,154.870
C06834=1085.032,421.813,394.815,177.451,28.757,154.867
C06835=1085.025,421.567,394.858,177.447,28.746,154.865
C06836=1085.018,421.320,394.900,177.443,28.735,154.863
C06837=1085.010,421.074,394.942,177.439,28.725,154.860
C06838=1085.004,420.829,394.985,177.435,28.714,154.858
C06839=1084.997,420.583,395.027,177.431,28.704,154.856
C06840=1084.990,420.336,395.070,177.426,28.693,154.854
C06841=1084.984,420.090,395.112,177.423,28.683,154.851
C06842=1084.977,419.844,395.155,177.419,28.672,154.849
C06843=1084.970,419.597,395.197,177.414,28.662,154.847
C06844=1084.963,419.350,395.239,177.410,28.651,154.845
C06845=1084.956,419.104,395.282,177.406,28.641,154.843
C06846=1084.950,418.858,395.323,177.402,28.631,154.840
C06847=1084.944,418.612,395.366,177.398,28.621,154.838
C06848=1084.937,418.365,395.408,177.394,28.611,154.836
C06849=1084.930,418.119,395.450,177.390,28.600,154.834
C06850=1084.923,417.873,395.492,177.386,28.590,154.832
C06851=1084.917,417.626,395.533,177.382,28.580,154.830
C06852=1084.910,417.380,395.576,177.378,28.569,154.827
C06853=1084.903,417.134,395.618,177.374,28.559,154.825
C06854=1084.897,416.888,395.660,177.370,28.550,154.823
C06855=1084.890,416.641,395.702,177.366,28.539,154.821
C06856=1084.884,416.394,395.744,177.362,28.530,154.819
C06857=1084.877,416.149,395.785,177.358,28.519,154.817
C06858=1084.870,415.902,395.828,177.354,28.509,154.815
C06859=1084.864,415.655,395.870,177.350,28.499,154.813
C06860=1084.856,415.409,395.911,177.346,28.489,154.811
C06861=1084.850,415.163,395.952,177.342,28.480,154.808
C06862=1084.843,414.916,395.995,177.338,28.470,154.806
C06863=1084.836,414.670,396.036,177.335,28.460,154.804
C06864=1084.830,414.423,396.077,177.330,28.450,154.802
C06865=1084.823,414.177,396.119,177.327,28.441,154.800
C06866=1084.816,413.930,396.160,177.322,28.431,154.798
C06867=1084.810,413.684,396.203,177.318,28.422,154.796
C06868=1084.803,413.438,396.244,177.315,28.412,154.794
C06869=1084.797,413.192,396.285,177.310,28.402,154.792
C06870=1084.790,412.945,396.327,177.307,28.393,154.790
C06871=1084.783,412.712,396.365,177.303,28.384,154.788
C06872=1084.778,412.478,396.405,177.300,28.375,154.787
C06873=1084.771,412.246,396.444,177.295,28.366,154.785
C06874=1084.764,412.011,396.483,177.292,28.357,154.783
C06875=1084.758,411.778,396.523,177.288,28.348,154.781
C06876=1084.752,411.545,396.561,177.285,28.339,154.779
C06877=1084.746,411.312,396.601,177.281,28.330,154.777
C06878=1084.739,411.079,396.639,177.278,28.321,154.775
C06879=1084.733,410.833,396.681,177.273,28.312,154.773
C06880=1084.726,410.586,396.722,177.270,28.303,154.772
C06881=1084.720,410.339,396.763,177.265,28.293,154.770
C06882=1084.713,410.092,396.804,177.262,28.284,154.768
C06883=1084.707,409.846,396.845,177.259,28.275,154.766
C06884=1084.700,409.599,396.886,177.254,28.265,154.764
C06885=1084.694,409.353,396.927,177.251,28.256,154.762
C06886=1084.687,409.106,396.968,177.246,28.247,154.760
C06887=1084.681,408.859,397.009,177.243,28.238,154.758
C06888=1084.675,408.614,397.050,177.239,28.229,154.756
C06889=1084.667,408.367,397.091,177.235,28.220,154.754
C06890=1084.662,408.120,397.132,177.232,28.211,154.753
C06891=1084.655,407.874,397.173,177.228,28.202,154.751
C06892=1084.649,407.627,397.214,177.224,28.193,154.749
C06893=1084.642,407.381,397.255,177.220,28.183,154.747
C06894=1084.636,407.134,397.295,177.217,28.175,154.745
C06895=1084.629,406.887,397.335,177.212,28.166,154.743
C06896=1084.623,406.641,397.377,177.209,28.157,154.742
C06897=1084.616,406.394,397.417,177.206,28.148,154.740
C06898=1084.609,406.147,397.458,177.202,28.139,154.738
C06899=1084.603,405.901,397.498,177.198,28.130,154.736
C06900=1084.597,405.654,397.539,177.194,28.121,154.734
C06901=1084.590,405.407,397.580,177.191,28.113,154.732
C06902=1084.583,405.161,397.621,177.187,28.104,154.731
C06903=1084.577,404.915,397.661,177.183,28.095,154.729
C06904=1084.571,404.668,397.701,177.179,28.087,154.727
C06905=1084.564,404.421,397.741,177.176,28.078,154.725
C06906=1084.558,404.174,397.782,177.172,28.069,154.724
C06907=1084.552,403.928,397.822,177.168,28.061,154.722
C06908=1084.545,403.681,397.862,177.164,28.052,154.720
C06909=1084.538,403.435,397.904,177.161,28.044,154.718
C06910=1084.532,403.188,397.944,177.157,28.035,154.717
C06911=1084.525,402.942,397.984,177.154,28.027,154.715
C06912=1084.519,402.695,398.024,177.149,28.018,154.713
C06913=1084.512,402.449,398.064,177.146,28.010,154.711
C06914=1084.505,402.201,398.105,177.142,28.001,154.710
C06915=1084.499,401.954,398.144,177.139,27.993,154.708
C06916=1084.493,401.708,398.184,177.135,27.985,154.706
C06917=1084.487,401.461,398.225,177.132,27.976,154.705
C06918=1084.480,401.215,398.265,177.127,27.968,154.703
C06919=1084.474,400.968,398.305,177.124,27.959,154.701
C06920=1084.468,400.722,398.345,177.121,27.951,154.700
C06921=1084.461,400.475,398.385,177.117,27.943,154.698
C06922=1084.454,400.228,398.424,177.113,27.935,154.696
C06923=1084.447,399.981,398.464,177.110,27.927,154.695
C06924=1084.441,399.735,398.505,177.106,27.918,154.693
C06925=1084.435,399.487,398.544,177.103,27.910,154.691
C06926=1084.429,399.241,398.584,177.099,27.901,154.690
C06927=1084.422,399.009,398.622,177.096,27.894,154.688
C06928=1084.417,398.777,398.660,177.092,27.887,154.687
C06929=1084.411,398.544,398.697,177.089,27.879,154.685
C06930=1084.405,398.311,398.734,177.085,27.871,154.684
C06931=1084.398,398.079,398.771,177.082,27.864,154.682
C06932=1084.392,397.847,398.809,177.079,27.856,154.681
C06933=1084.386,397.615,398.846,177.075,27.848,154.679
C06934=1084.380,397.382,398.883,177.072,27.841,154.678
C06935=1084.374,397.135,398.923,177.068,27.833,154.676
C06936=1084.368,396.888,398.963,177.065,27.825,154.675
C06937=1084.361,396.641,399.003,177.061,27.817,154.673
C06938=1084.354,396.395,399.042,177.058,27.809,154.671
C06939=1084.348,396.148,399.082,177.054,27.802,154.670
C06940=1084.342,395.901,399.121,177.050,27.794,154.668
C06941=1084.336,395.655,399.160,177.047,27.786,154.667
C06942=1084.329,395.408,399.200,177.043,27.778,154.665
C06943=1084.323,395.161,399.239,177.040,27.770,154.664
C06944=1084.316,394.914,399.278,177.036,27.762,154.662
C06945=1084.310,394.668,399.318,177.033,27.755,154.661
C06946=1084.304,394.421,399.358,177.029,27.747,154.659
C06947=1084.297,394.174,399.396,177.026,27.739,154.658
C06948=1084.291,393.927,399.436,177.022,27.731,154.656
C06949=1084.285,393.681,399.474,177.019,27.724,154.655
C06950=1084.279,393.434,399.515,177.015,27.716,154.653
C06951=1084.272,393.187,399.553,177.011,27.708,154.651
C06952=1084.266,392.940,399.593,177.008,27.701,154.650
C06953=1084.259,392.693,399.632,177.004,27.693,154.649
C06954=1084.253,392.447,399.671,177.001,27.686,154.647
C06955=1084.247,392.200,399.710,176.997,27.678,154.646
C06956=1084.240,391.953,399.749,176.994,27.670,154.644
C06957=1084.234,391.706,399.788,176.990,27.663,154.643
C06958=1084.228,391.460,399.827,176.987,27.655,154.641
C06959=1084.221,391.213,399.866,176.983,27.648,154.640
C06960=1084.215,390.966,399.905,176.979,27.640,154.638
C06961=1084.208,390.719,399.943,176.976,27.633,154.637
C06962=1084.202,390.473,399.982,176.973,27.626,154.635
C06963=1084.195,390.226,400.021,176.969,27.619,154.634
C06964=1084.189,389.979,400.059,176.966,27.611,154.633
C06965=1084.183,389.731,400.099,176.962,27.604,154.631
C06966=1084.177,389.485,400.137,176.959,27.597,154.630
C06967=1084.170,389.238,400.176,176.955,27.589,154.628
C06968=1084.163,388.992,400.215,176.952,27.582,154.627
C06969=1084.158,388.745,400.253,176.948,27.574,154.626
C06970=1084.151,388.498,400.292,176.944,27.567,154.624
C06971=1084.144,388.251,400.331,176.941,27.560,154.623
C06972=1084.138,388.004,400.369,176.937,27.553,154.621
C06973=1084.132,387.757,400.408,176.934,27.545,154.620
C06974=1084.126,387.511,400.447,176.931,27.538,154.619
C06975=1084.120,387.263,400.485,176.927,27.531,154.617
C06976=1084.113,387.017,400.524,176.924,27.524,154.616
C06977=1084.107,386.771,400.562,176.920,27.517,154.614
C06978=1084.101,386.523,400.601,176.917,27.510,154.613
C06979=1084.095,386.277,400.639,176.913,27.502,154.612
C06980=1084.088,386.029,400.677,176.909,27.495,154.610
C06981=1084.082,385.783,400.716,176.907,27.488,154.609
C06982=1084.075,385.536,400.754,176.903,27.481,154.608
C06983=1084.070,385.310,400.789,176.899,27.475,154.607
C06984=1084.064,385.084,400.825,176.897,27.468,154.605
C06985=1084.059,384.859,400.859,176.893,27.462,154.604
C06986=1084.053,384.633,400.894,176.890,27.455,154.603
C06987=1084.047,384.408,400.929,176.887,27.449,154.602
C06988=1084.041,384.183,400.964,176.884,27.443,154.600
C06989=1084.036,383.957,400.999,176.881,27.437,154.599
C06990=1084.031,383.732,401.034,176.877,27.430,154.598
C06991=1084.024,383.485,401.073,176.875,27.423,154.597
C06992=1084.018,383.238,401.110,176.871,27.416,154.595
C06993=1084.012,382.991,401.148,176.867,27.409,154.594
C06994=1084.006,382.744,401.186,176.864,27.402,154.593
C06995=1083.999,382.497,401.225,176.860,27.395,154.592
C06996=1083.993,382.251,401.263,176.857,27.389,154.590
C06997=1083.986,382.003,401.301,176.854,27.382,154.589
C06998=1083.981,381.756,401.339,176.850,27.375,154.588
C06999=1083.975,381.510,401.376,176.846,27.368,154.586
C07000=1083.968,381.262,401.415,176.844,27.361,154.585
C07001=1083.962,381.015,401.452,176.840,27.355,154.584
C07002=1083.955,380.768,401.490,176.836,27.348,154.583
C07003=1083.949,380.522,401.528,176.833,27.341,154.581
C07004=1083.943,380.274,401.566,176.830,27.335,154.580
C07005=1083.937,380.027,401.603,176.826,27.328,154.579
C07006=1083.931,379.781,401.641,176.823,27.322,154.578
C07007=1083.924,379.533,401.679,176.819,27.315,154.576
C07008=1083.918,379.287,401.716,176.817,27.308,154.575
C07009=1083.912,379.040,401.754,176.813,27.302,154.574
C07010=1083.905,378.793,401.792,176.809,27.295,154.573
C07011=1083.899,378.546,401.830,176.806,27.288,154.571
C07012=1083.893,378.298,401.868,176.803,27.282,154.570
C07013=1083.887,378.051,401.905,176.799,27.275,154.569
C07014=1083.881,377.805,401.942,176.795,27.269,154.568
C07015=1083.874,377.517,401.986,176.792,27.261,154.566
C07016=1083.866,377.229,402.030,176.788,27.253,154.565
C07017=1083.859,376.942,402.074,176.784,27.246,154.564
C07018=1083.851,376.654,402.118,176.780,27.238,154.562
C07019=1083.845,376.407,402.155,176.777,27.232,154.561
C07020=1083.840,376.159,402.192,176.773,27.225,154.560
C07021=1083.833,375.913,402.229,176.770,27.219,154.559
C07022=1083.827,375.666,402.267,176.767,27.212,154.557
C07023=1083.821,375.418,402.305,176.763,27.206,154.556
C07024=1083.815,375.171,402.342,176.760,27.199,154.555
C07025=1083.809,374.924,402.379,176.757,27.193,154.554
C07026=1083.803,374.678,402.417,176.753,27.187,154.553
C07027=1083.797,374.430,402.454,176.749,27.180,154.552
C07028=1083.790,374.183,402.491,176.747,27.174,154.550
C07029=1083.785,373.936,402.528,176.743,27.168,154.549
C07030=1083.779,373.689,402.566,176.739,27.161,154.548
C07031=1083.772,373.442,402.602,176.737,27.155,154.547
C07032=1083.766,373.195,402.641,176.733,27.149,154.546
C07033=1083.759,372.948,402.677,176.729,27.143,154.545
C07034=1083.754,372.700,402.714,176.726,27.136,154.544
C07035=1083.747,372.454,402.751,176.723,27.130,154.542
C07036=1083.741,372.207,402.788,176.720,27.124,154.541
C07037=1083.735,371.959,402.825,176.716,27.118,154.540
C07038=1083.728,371.712,402.862,176.713,27.112,154.539
C07039=1083.719,371.330,402.919,176.708,27.102,154.537
C07040=1083.709,370.948,402.976,176.703,27.093,154.536
C07041=1083.700,370.566,403.033,176.697,27.083,154.534
C07042=1083.690,370.184,403.090,176.692,27.074,154.532
C07043=1083.684,369.937,403.127,176.689,27.067,154.531
C07044=1083.678,369.690,403.164,176.686,27.062,154.530
C07045=1083.672,369.442,403.201,176.682,27.056,154.529
C07046=1083.666,369.195,403.237,176.679,27.049,154.528
C07047=1083.660,368.948,403.274,176.676,27.043,154.527
C07048=1083.654,368.701,403.311,176.672,27.037,154.526
C07049=1083.648,368.454,403.347,176.669,27.031,154.525
C07050=1083.642,368.207,403.384,176.666,27.025,154.524
C07051=1083.636,367.959,403.421,176.663,27.020,154.523
C07052=1083.630,367.712,403.457,176.659,27.014,154.522
C07053=1083.623,367.465,403.494,176.655,27.007,154.520
C07054=1083.618,367.218,403.531,176.653,27.001,154.519
C07055=1083.611,366.971,403.567,176.649,26.995,154.518
C07056=1083.605,366.724,403.603,176.646,26.990,154.517
C07057=1083.599,366.476,403.640,176.642,26.984,154.516
C07058=1083.593,366.229,403.677,176.639,26.978,154.515
C07059=1083.587,365.982,403.713,176.636,26.972,154.514
C07060=1083.581,365.734,403.750,176.633,26.966,154.513
C07061=1083.575,365.487,403.786,176.629,26.960,154.512
C07062=1083.569,365.240,403.823,176.626,26.954,154.511
C07063=1083.562,364.993,403.859,176.623,26.948,154.510
C07064=1083.556,364.746,403.895,176.620,26.943,154.509
C07065=1083.551,364.498,403.932,176.616,26.937,154.508
C07066=1083.544,364.251,403.968,176.613,26.931,154.507
C07067=1083.538,364.003,404.004,176.610,26.925,154.506
C07068=1083.532,363.756,404.040,176.606,26.919,154.505
C07069=1083.526,363.509,404.077,176.603,26.914,154.504
C07070=1083.520,363.262,404.112,176.599,26.907,154.503
C07071=1083.514,363.015,404.149,176.597,26.902,154.502
C07072=1083.508,362.768,404.185,176.593,26.896,154.501
C07073=1083.502,362.521,404.221,176.590,26.891,154.500
C07074=1083.495,362.274,404.257,176.586,26.885,154.499
C07075=1083.489,362.026,404.293,176.583,26.879,154.498
C07076=1083.483,361.779,404.329,176.581,26.873,154.497
C07077=1083.477,361.531,404.365,176.577,26.868,154.496
C07078=1083.471,361.284,404.402,176.574,26.862,154.495
C07079=1083.465,361.037,404.437,176.570,26.857,154.494
C07080=1083.459,360.789,404.473,176.567,26.851,154.493
C07081=1083.453,360.542,404.510,176.564,26.845,154.492
C07082=1083.447,360.295,404.545,176.561,26.840,154.491
C07083=1083.440,360.048,404.581,176.557,26.834,154.490
C07084=1083.434,359.800,404.617,176.554,26.828,154.489
C07085=1083.429,359.553,404.652,176.550,26.823,154.488
C07086=1083.423,359.305,404.688,176.548,26.818,154.487
C07087=1083.417,359.058,404.725,176.544,26.811,154.486
C07088=1083.411,358.811,404.760,176.541,26.806,154.485
C07089=1083.404,358.563,404.796,176.538,26.801,154.484
C07090=1083.399,358.316,404.831,176.534,26.795,154.483
C07091=1083.388,357.909,404.891,176.529,26.786,154.482
C07092=1083.378,357.502,404.949,176.524,26.778,154.480
C07093=1083.368,357.095,405.008,176.518,26.768,154.479
C07094=1083.358,356.688,405.066,176.513,26.759,154.477
C07095=1083.352,356.442,405.102,176.510,26.754,154.476
C07096=1083.346,356.194,405.138,176.507,26.748,154.475
C07097=1083.340,355.947,405.173,176.504,26.743,154.475
C07098=1083.335,355.700,405.209,176.500,26.738,154.474
C07099=1083.328,355.452,405.244,176.497,26.732,154.473
C07100=1083.322,355.205,405.280,176.494,26.727,154.472
C07101=1083.317,354.958,405.315,176.490,26.721,154.471
C07102=1083.311,354.710,405.351,176.488,26.716,154.470
C07103=1083.304,354.462,405.386,176.484,26.710,154.469
C07104=1083.299,354.215,405.420,176.481,26.705,154.468
C07105=1083.293,353.967,405.456,176.478,26.700,154.467
C07106=1083.287,353.720,405.492,176.474,26.695,154.466
C07107=1083.280,353.473,405.527,176.471,26.689,154.465
C07108=1083.274,353.225,405.562,176.468,26.684,154.464
C07109=1083.268,352.978,405.598,176.465,26.678,154.464
C07110=1083.262,352.731,405.633,176.462,26.673,154.463
C07111=1083.256,352.483,405.668,176.458,26.668,154.462
C07112=1083.250,352.235,405.704,176.455,26.663,154.461
C07113=1083.244,351.988,405.738,176.452,26.658,154.460
C07114=1083.238,351.741,405.774,176.449,26.652,154.459
C07115=1083.232,351.493,405.808,176.446,26.647,154.458
C07116=1083.226,351.246,405.844,176.443,26.642,154.457
C07117=1083.220,350.998,405.879,176.439,26.636,154.457
C07118=1083.214,350.751,405.914,176.436,26.632,154.456
C07119=1083.208,350.503,405.949,176.433,26.626,154.455
C07120=1083.202,350.256,405.984,176.429,26.621,154.454
C07121=1083.196,350.008,406.019,176.427,26.616,154.453
C07122=1083.190,349.761,406.054,176.424,26.611,154.452
C07123=1083.184,349.513,406.088,176.420,26.605,154.451
C07124=1083.178,349.266,406.124,176.417,26.600,154.451
C07125=1083.172,349.018,406.158,176.414,26.595,154.450
C07126=1083.166,348.771,406.194,176.410,26.590,154.449
C07127=1083.160,348.524,406.228,176.407,26.585,154.448
C07128=1083.154,348.276,406.264,176.405,26.580,154.447
C07129=1083.148,348.029,406.298,176.401,26.575,154.446
C07130=1083.142,347.781,406.334,176.398,26.569,154.445
C07131=1083.136,347.534,406.368,176.395,26.565,154.445
C07132=1083.130,347.286,406.403,176.391,26.559,154.444
C07133=1083.124,347.039,406.437,176.388,26.554,154.443
C07134=1083.118,346.791,406.472,176.385,26.549,154.442
C07135=1083.113,346.544,406.507,176.382,26.545,154.441
C07136=1083.106,346.296,406.542,176.379,26.539,154.440
C07137=1083.101,346.048,406.576,176.376,26.534,154.440
C07138=1083.094,345.801,406.611,176.373,26.529,154.439
C07139=1083.088,345.553,406.645,176.369,26.524,154.438
C07140=1083.083,345.305,406.680,176.366,26.519,154.437
C07141=1083.077,345.058,406.714,176.363,26.514,154.436
C07142=1083.071,344.811,406.749,176.360,26.509,154.436
C07143=1083.061,344.407,406.805,176.355,26.501,154.434
C07144=1083.052,344.003,406.862,176.350,26.493,154.433
C07145=1083.041,343.599,406.918,176.345,26.485,154.432
C07146=1083.031,343.195,406.974,176.339,26.477,154.430
C07147=1083.026,342.948,407.008,176.337,26.472,154.430
C07148=1083.019,342.700,407.043,176.333,26.467,154.429
C07149=1083.014,342.453,407.077,176.330,26.462,154.428
C07150=1083.008,342.205,407.112,176.327,26.457,154.427
C07151=1083.002,341.957,407.146,176.324,26.452,154.426
C07152=1082.996,341.710,407.180,176.320,26.447,154.426
C07153=1082.989,341.462,407.214,176.317,26.442,154.425
C07154=1082.983,341.215,407.248,176.314,26.438,154.424
C07155=1082.978,340.967,407.282,176.311,26.433,154.423
C07156=1082.972,340.719,407.317,176.307,26.428,154.422
C07157=1082.966,340.472,407.351,176.305,26.423,154.422
C07158=1082.960,340.225,407.385,176.302,26.419,154.421
C07159=1082.954,339.977,407.420,176.299,26.414,154.420
C07160=1082.948,339.729,407.453,176.296,26.409,154.419
C07161=1082.942,339.481,407.487,176.292,26.404,154.419
C07162=1082.936,339.234,407.521,176.289,26.399,154.418
C07163=1082.930,338.986,407.556,176.286,26.394,154.417
C07164=1082.924,338.739,407.590,176.283,26.389,154.416
C07165=1082.919,338.491,407.623,176.280,26.384,154.416
C07166=1082.913,338.243,407.658,176.276,26.380,154.415
C07167=1082.907,337.995,407.692,176.273,26.375,154.414
C07168=1082.900,337.748,407.726,176.270,26.370,154.413
C07169=1082.895,337.500,407.759,176.267,26.366,154.413
C07170=1082.888,337.252,407.793,176.265,26.361,154.412
C07171=1082.882,337.005,407.827,176.261,26.356,154.411
C07172=1082.877,336.757,407.861,176.258,26.352,154.410
C07173=1082.871,336.510,407.895,176.255,26.347,154.410
C07174=1082.865,336.262,407.929,176.252,26.342,154.409
C07175=1082.859,336.014,407.963,176.249,26.338,154.408
C07176=1082.853,335.767,407.997,176.246,26.333,154.407
C07177=1082.848,335.519,408.030,176.242,26.328,154.407
C07178=1082.840,335.271,408.064,176.239,26.323,154.406
C07179=1082.835,335.023,408.097,176.236,26.318,154.405
C07180=1082.829,334.776,408.131,176.233,26.314,154.405
C07181=1082.823,334.528,408.164,176.230,26.309,154.404
C07182=1082.818,334.281,408.199,176.227,26.305,154.403
C07183=1082.812,334.033,408.232,176.224,26.300,154.402
C07184=1082.806,333.785,408.266,176.220,26.295,154.402
C07185=1082.799,333.537,408.299,176.218,26.291,154.401
C07186=1082.793,333.290,408.333,176.215,26.286,154.400
C07187=1082.788,333.042,408.366,176.212,26.281,154.399
C07188=1082.782,332.794,408.400,176.209,26.277,154.399
C07189=1082.776,332.547,408.434,176.206,26.272,154.398
C07190=1082.770,332.299,408.467,176.203,26.268,154.397
C07191=1082.765,332.052,408.500,176.200,26.263,154.397
C07192=1082.759,331.804,408.534,176.196,26.258,154.396
C07193=1082.753,331.556,408.568,176.193,26.254,154.395
C07194=1082.746,331.308,408.600,176.190,26.249,154.394
C07195=1082.737,330.899,408.656,176.185,26.242,154.393
C07196=1082.726,330.489,408.710,176.180,26.235,154.392
C07197=1082.717,330.080,408.766,176.175,26.227,154.391
C07198=1082.706,329.671,408.820,176.170,26.220,154.390
C07199=1082.701,329.423,408.853,176.167,26.215,154.389
C07200=1082.694,329.175,408.886,176.164,26.211,154.389
C07201=1082.688,328.928,408.920,176.161,26.207,154.388
C07202=1082.682,328.680,408.953,176.158,26.202,154.387
C07203=1082.677,328.432,408.986,176.155,26.198,154.387
C07204=1082.670,328.185,409.019,176.152,26.194,154.386
C07205=1082.664,327.936,409.053,176.148,26.189,154.385
C07206=1082.658,327.689,409.085,176.145,26.185,154.385
C07207=1082.652,327.441,409.119,176.142,26.180,154.384
C07208=1082.646,327.193,409.152,176.139,26.176,154.383
C07209=1082.640,326.945,409.185,176.136,26.171,154.383
C07210=1082.634,326.698,409.218,176.133,26.167,154.382
C07211=1082.628,326.450,409.250,176.130,26.162,154.381
C07212=1082.622,326.202,409.284,176.127,26.158,154.381
C07213=1082.616,325.954,409.316,176.124,26.154,154.380
C07214=1082.611,325.707,409.350,176.121,26.149,154.379
C07215=1082.605,325.458,409.382,176.118,26.145,154.379
C07216=1082.599,325.210,409.415,176.115,26.140,154.378
C07217=1082.593,324.964,409.447,176.112,26.136,154.377
C07218=1082.587,324.716,409.480,176.109,26.132,154.377
C07219=1082.581,324.468,409.514,176.106,26.127,154.376
C07220=1082.575,324.220,409.546,176.103,26.123,154.375
C07221=1082.570,323.972,409.579,176.100,26.119,154.375
C07222=1082.564,323.724,409.612,176.097,26.114,154.374
C07223=1082.557,323.477,409.644,176.094,26.110,154.373
C07224=1082.552,323.229,409.678,176.091,26.106,154.373
C07225=1082.546,322.981,409.710,176.088,26.102,154.372
C07226=1082.539,322.733,409.743,176.085,26.097,154.372
C07227=1082.534,322.485,409.776,176.081,26.093,154.371
C07228=1082.528,322.238,409.808,176.078,26.088,154.370
C07229=1082.522,321.990,409.840,176.075,26.084,154.370
C07230=1082.517,321.742,409.874,176.072,26.080,154.369
C07231=1082.511,321.494,409.906,176.069,26.075,154.368
C07232=1082.504,321.246,409.938,176.066,26.071,154.368
C07233=1082.499,320.998,409.972,176.063,26.066,154.367
C07234=1082.493,320.751,410.003,176.060,26.062,154.366
C07235=1082.487,320.503,410.036,176.057,26.058,154.366
C07236=1082.482,320.255,410.069,176.054,26.054,154.365
C07237=1082.476,320.007,410.101,176.051,26.049,154.364
C07238=1082.470,319.760,410.133,176.048,26.045,154.364
C07239=1082.464,319.512,410.166,176.046,26.041,154.363
C07240=1082.459,319.264,410.199,176.043,26.037,154.362
C07241=1082.452,319.016,410.231,176.040,26.032,154.362
C07242=1082.447,318.768,410.263,176.037,26.028,154.361
C07243=1082.441,318.521,410.296,176.034,26.024,154.361
C07244=1082.435,318.272,410.328,176.031,26.020,154.360
C07245=1082.429,318.025,410.361,176.028,26.015,154.359
C07246=1082.424,317.777,410.393,176.025,26.011,154.359
C07247=1082.414,317.361,410.448,176.020,26.004,154.358
C07248=1082.404,316.945,410.501,176.015,25.997,154.357
C07249=1082.395,316.528,410.556,176.010,25.990,154.355
C07250=1082.385,316.113,410.610,176.005,25.982,154.354
C07251=1082.379,315.865,410.642,176.002,25.978,154.354
C07252=1082.374,315.617,410.674,175.999,25.974,154.353
C07253=1082.369,315.369,410.706,175.996,25.969,154.353
C07254=1082.362,315.121,410.739,175.993,25.965,154.352
C07255=1082.356,314.873,410.771,175.990,25.961,154.351
C07256=1082.351,314.626,410.802,175.987,25.957,154.351
C07257=1082.345,314.377,410.834,175.984,25.953,154.350
C07258=1082.339,314.129,410.867,175.982,25.949,154.350
C07259=1082.333,313.881,410.899,175.979,25.945,154.349
C07260=1082.327,313.634,410.930,175.976,25.941,154.348
C07261=1082.321,313.386,410.962,175.973,25.937,154.348
C07262=1082.315,313.138,410.994,175.970,25.933,154.347
C07263=1082.309,312.891,411.026,175.967,25.928,154.347
C07264=1082.303,312.642,411.058,175.964,25.925,154.346
C07265=1082.297,312.394,411.089,175.961,25.921,154.346
C07266=1082.291,312.147,411.121,175.958,25.916,154.345
C07267=1082.285,311.899,411.153,175.955,25.912,154.344
C07268=1082.279,311.650,411.185,175.952,25.909,154.344
C07269=1082.273,311.403,411.216,175.949,25.904,154.343
C07270=1082.267,311.155,411.248,175.946,25.900,154.343
C07271=1082.262,310.908,411.280,175.943,25.896,154.342
C07272=1082.256,310.659,411.312,175.941,25.892,154.341
C07273=1082.249,310.411,411.343,175.937,25.888,154.341
C07274=1082.244,310.164,411.375,175.935,25.884,154.340
C07275=1082.238,309.916,411.407,175.931,25.880,154.340
C07276=1082.231,309.668,411.438,175.928,25.876,154.339
C07277=1082.226,309.420,411.469,175.925,25.872,154.339
C07278=1082.220,309.172,411.501,175.922,25.868,154.338
C07279=1082.214,308.924,411.533,175.919,25.864,154.338
C07280=1082.208,308.676,411.565,175.916,25.860,154.337
C07281=1082.202,308.429,411.596,175.913,25.856,154.336
C07282=1082.196,308.180,411.628,175.911,25.852,154.336
C07283=1082.190,307.932,411.659,175.908,25.848,154.335
C07284=1082.185,307.684,411.691,175.905,25.844,154.335
C07285=1082.179,307.437,411.722,175.902,25.840,154.334
